LIN {X 0,Y 625.724,Z 847.824,A -85,B 0,C 180,E1 -6603.018,E2 -6603.018} C_VEL
LIN {X 0,Y 627.181,Z 825.978,A -85,B 0,C 180,E1 -6603.807,E2 -6603.807} C_VEL
LIN {X 0,Y 628.649,Z 801.844,A -85,B 0,C 180,E1 -6604.509,E2 -6604.509} C_VEL
LIN {X 0,Y 629.711,Z 779.175,A -85,B 0,C 180,E1 -6605.002,E2 -6605.002} C_VEL
LIN {X 0,Y 630.485,Z 755.504,A -85,B 0,C 180,E1 -6605.381,E2 -6605.381} C_VEL
LIN {X 0,Y 634.655,Z 505.847,A -85,B 0,C 180,E1 -6608.568,E2 -6608.568} C_VEL
LIN {X 0,Y 636.212,Z 410.489,A -85,B 0,C 180,E1 -6609.813,E2 -6609.813} C_VEL
LIN {X 0,Y 632.38,Z 394.65,A -85,B 0,C 180,E1 -6610.331,E2 -6610.331} C_VEL
LIN {X 0,Y 620.426,Z 374.094,A -85,B 0,C 180,E1 -6611.604,E2 -6611.604} C_VEL
LIN {X 0,Y 613.158,Z 355.776,A -85,B 0,C 180,E1 -6613.881,E2 -6613.881} C_VEL
LIN {X 0,Y 609.05,Z 345.363,A -85,B 0,C 180,E1 -6615.266,E2 -6615.266} C_VEL
LIN {X 0,Y 609.013,Z 345.362,A -85,B 0,C 180,E1 -6618.196,E2 -6618.196} C_VEL
LIN {X 0,Y 609.063,Z 345.362,A -85,B 0,C 180,E1 -6621.282,E2 -6621.282} C_VEL
LIN {X 0,Y 609.006,Z 345.32,A -85,B 0,C 180,E1 -6624.232,E2 -6624.232} C_VEL
LIN {X 0,Y 609.058,Z 345.363,A -85,B 0,C 180,E1 -6627.42,E2 -6627.42} C_VEL
LIN {X 0,Y 609.014,Z 345.363,A -85,B 0,C 180,E1 -6630.384,E2 -6630.384} C_VEL
LIN {X 0,Y 609.063,Z 345.359,A -85,B 0,C 180,E1 -6633.478,E2 -6633.478} C_VEL
LIN {X 0,Y 609.014,Z 345.358,A -85,B 0,C 180,E1 -6636.487,E2 -6636.487} C_VEL
LIN {X 0,Y 609.057,Z 345.353,A -85,B 0,C 180,E1 -6639.632,E2 -6639.632} C_VEL
LIN {X 0,Y 609.015,Z 345.363,A -85,B 0,C 180,E1 -6642.614,E2 -6642.614} C_VEL
LIN {X 0,Y 609.06,Z 345.366,A -85,B 0,C 180,E1 -6645.744,E2 -6645.744} C_VEL
LIN {X 0,Y 609.015,Z 345.354,A -85,B 0,C 180,E1 -6648.733,E2 -6648.733} C_VEL
LIN {X 0,Y 609.056,Z 345.352,A -85,B 0,C 180,E1 -6651.883,E2 -6651.883} C_VEL
LIN {X 0,Y 609.017,Z 345.364,A -85,B 0,C 180,E1 -6654.819,E2 -6654.819} C_VEL
LIN {X 0,Y 609.05,Z 345.354,A -85,B 0,C 180,E1 -6658.024,E2 -6658.024} C_VEL
LIN {X 0,Y 609.018,Z 345.36,A -85,B 0,C 180,E1 -6660.962,E2 -6660.962} C_VEL
LIN {X 0,Y 609.05,Z 345.368,A -85,B 0,C 180,E1 -6664.142,E2 -6664.142} C_VEL
LIN {X 0,Y 609.017,Z 345.351,A -85,B 0,C 180,E1 -6667.073,E2 -6667.073} C_VEL
LIN {X 0,Y 609.043,Z 345.356,A -85,B 0,C 180,E1 -6670.309,E2 -6670.309} C_VEL
LIN {X 0,Y 609.027,Z 345.363,A -85,B 0,C 180,E1 -6673.288,E2 -6673.288} C_VEL
LIN {X 0,Y 609.029,Z 345.361,A -85,B 0,C 180,E1 -6676.599,E2 -6676.599} C_VEL
LIN {X 0,Y 609.043,Z 345.358,A -85,B 0,C 180,E1 -6679.567,E2 -6679.567} C_VEL
LIN {X 0,Y 609.023,Z 345.362,A -85,B 0,C 180,E1 -6682.797,E2 -6682.797} C_VEL
LIN {X 0,Y 609.053,Z 345.361,A -85,B 0,C 180,E1 -6685.789,E2 -6685.789} C_VEL
LIN {X 0,Y 609.022,Z 345.367,A -85,B 0,C 180,E1 -6688.969,E2 -6688.969} C_VEL
LIN {X 0,Y 609.056,Z 345.351,A -85,B 0,C 180,E1 -6691.923,E2 -6691.923} C_VEL
LIN {X 0,Y 609.021,Z 345.362,A -85,B 0,C 180,E1 -6695.074,E2 -6695.074} C_VEL
LIN {X 0,Y 609.07,Z 345.352,A -85,B 0,C 180,E1 -6698.154,E2 -6698.154} C_VEL
LIN {X 0,Y 609.02,Z 345.37,A -85,B 0,C 180,E1 -6701.301,E2 -6701.301} C_VEL
LIN {X 0,Y 609.078,Z 345.362,A -85,B 0,C 180,E1 -6704.429,E2 -6704.429} C_VEL
LIN {X 0,Y 609.068,Z 345.578,A -85,B 0,C 180,E1 -6707.031,E2 -6707.031} C_VEL
LIN {X 0,Y 611.046,Z 350.8,A -85,B 0,C 180,E1 -6707.701,E2 -6707.701} C_VEL
LIN {X 0,Y 624.951,Z 372.362,A -85,B 0,C 180,E1 -6709.181,E2 -6709.181} C_VEL
LIN {X 0,Y 636.425,Z 391.644,A -85,B 0,C 180,E1 -6710.353,E2 -6710.353} C_VEL
LIN {X 0,Y 635.55,Z 441.225,A -85,B 0,C 180,E1 -6710.999,E2 -6710.999} C_VEL
LIN {X 0,Y 634.674,Z 448.921,A -85,B 0,C 180,E1 -6711.044,E2 -6711.044} C_VEL
LIN {X 0,Y 629.403,Z 469.491,A -85,B 0,C 180,E1 -6710.95,E2 -6710.95} C_VEL
LIN {X 0,Y 628.688,Z 476.1,A -85,B 0,C 180,E1 -6710.992,E2 -6710.992} C_VEL
LIN {X 0,Y 624.153,Z 726.916,A -85,B 0,C 180,E1 -6714.229,E2 -6714.229} C_VEL
LIN {X 0,Y 623.344,Z 751.398,A -85,B 0,C 180,E1 -6714.622,E2 -6714.622} C_VEL
LIN {X 0,Y 622.243,Z 774.459,A -85,B 0,C 180,E1 -6715.131,E2 -6715.131} C_VEL
LIN {X 0,Y 620.781,Z 797.913,A -85,B 0,C 180,E1 -6715.825,E2 -6715.825} C_VEL
LIN {X 0,Y 619.291,Z 818.986,A -85,B 0,C 180,E1 -6716.594,E2 -6716.594} C_VEL
LIN {X 0,Y 617.333,Z 842.509,A -85,B 0,C 180,E1 -6717.635,E2 -6717.635} C_VEL
LIN {X 0,Y 615.596,Z 861.479,A -85,B 0,C 180,E1 -6718.629,E2 -6718.629} C_VEL
LIN {X 0,Y 613.582,Z 882.127,A -85,B 0,C 180,E1 -6719.873,E2 -6719.873} C_VEL
LIN {X 0,Y 611.515,Z 901.861,A -85,B 0,C 180,E1 -6721.268,E2 -6721.268} C_VEL
LIN {X 0,Y 609.523,Z 921.125,A -85,B 0,C 180,E1 -6722.815,E2 -6722.815} C_VEL
LIN {X 0,Y 607.551,Z 939.267,A -85,B 0,C 180,E1 -6724.509,E2 -6724.509} C_VEL
LIN {X 0,Y 605.872,Z 955.81,A -85,B 0,C 180,E1 -6726.254,E2 -6726.254} C_VEL
LIN {X 0,Y 604.297,Z 971.472,A -85,B 0,C 180,E1 -6728.164,E2 -6728.164} C_VEL
LIN {X 0,Y 602.991,Z 986.499,A -85,B 0,C 180,E1 -6730.228,E2 -6730.228} C_VEL
LIN {X 0,Y 601.969,Z 999.427,A -85,B 0,C 180,E1 -6732.304,E2 -6732.304} C_VEL
LIN {X 0,Y 601.21,Z 1010.682,A -85,B 0,C 180,E1 -6734.37,E2 -6734.37} C_VEL
LIN {X 0,Y 600.63,Z 1020.967,A -85,B 0,C 180,E1 -6736.621,E2 -6736.621} C_VEL
LIN {X 0,Y 600.302,Z 1028.497,A -85,B 0,C 180,E1 -6738.568,E2 -6738.568} C_VEL
LIN {X 0,Y 600.056,Z 1036.101,A -85,B 0,C 180,E1 -6740.988,E2 -6740.988} C_VEL
LIN {X 0,Y 599.974,Z 1041.005,A -85,B 0,C 180,E1 -6743.012,E2 -6743.012} C_VEL
LIN {X 0,Y 599.921,Z 1045.157,A -85,B 0,C 180,E1 -6745.316,E2 -6745.316} C_VEL
LIN {X 0,Y 599.899,Z 1047.463,A -85,B 0,C 180,E1 -6747.516,E2 -6747.516} C_VEL
LIN {X 0,Y 599.894,Z 1048.384,A -85,B 0,C 180,E1 -6749.523,E2 -6749.523} C_VEL
LIN {X 0,Y 599.908,Z 1047.935,A -85,B 0,C 180,E1 -6751.91,E2 -6751.91} C_VEL
LIN {X 0,Y 599.919,Z 1046.062,A -85,B 0,C 180,E1 -6754.014,E2 -6754.014} C_VEL
LIN {X 0,Y 599.948,Z 1042.77,A -85,B 0,C 180,E1 -6756.219,E2 -6756.219} C_VEL
LIN {X 0,Y 600.026,Z 1037.609,A -85,B 0,C 180,E1 -6758.529,E2 -6758.529} C_VEL
LIN {X 0,Y 600.186,Z 1032.047,A -85,B 0,C 180,E1 -6760.462,E2 -6760.462} C_VEL
LIN {X 0,Y 600.514,Z 1023.769,A -85,B 0,C 180,E1 -6762.794,E2 -6762.794} C_VEL
LIN {X 0,Y 600.963,Z 1014.847,A -85,B 0,C 180,E1 -6764.846,E2 -6764.846} C_VEL
LIN {X 0,Y 601.657,Z 1003.931,A -85,B 0,C 180,E1 -6767.007,E2 -6767.007} C_VEL
LIN {X 0,Y 602.568,Z 991.521,A -85,B 0,C 180,E1 -6769.081,E2 -6769.081} C_VEL
LIN {X 0,Y 603.644,Z 978.717,A -85,B 0,C 180,E1 -6770.964,E2 -6770.964} C_VEL
LIN {X 0,Y 605.162,Z 962.65,A -85,B 0,C 180,E1 -6773.027,E2 -6773.027} C_VEL
LIN {X 0,Y 606.722,Z 947.311,A -85,B 0,C 180,E1 -6774.761,E2 -6774.761} C_VEL
LIN {X 0,Y 608.619,Z 929.224,A -85,B 0,C 180,E1 -6776.543,E2 -6776.543} C_VEL
LIN {X 0,Y 610.398,Z 912.383,A -85,B 0,C 180,E1 -6778.001,E2 -6778.001} C_VEL
LIN {X 0,Y 612.623,Z 891.447,A -85,B 0,C 180,E1 -6779.58,E2 -6779.58} C_VEL
LIN {X 0,Y 614.454,Z 873.223,A -85,B 0,C 180,E1 -6780.772,E2 -6780.772} C_VEL
LIN {X 0,Y 616.495,Z 852.089,A -85,B 0,C 180,E1 -6781.978,E2 -6781.978} C_VEL
LIN {X 0,Y 618.343,Z 830.28,A -85,B 0,C 180,E1 -6783.021,E2 -6783.021} C_VEL
LIN {X 0,Y 620.188,Z 807.62,A -85,B 0,C 180,E1 -6783.934,E2 -6783.934} C_VEL
LIN {X 0,Y 621.651,Z 784.687,A -85,B 0,C 180,E1 -6784.673,E2 -6784.673} C_VEL
LIN {X 0,Y 622.771,Z 764.523,A -85,B 0,C 180,E1 -6785.194,E2 -6785.194} C_VEL
LIN {X 0,Y 623.81,Z 738.844,A -85,B 0,C 180,E1 -6785.687,E2 -6785.687} C_VEL
LIN {X 0,Y 626.912,Z 571.696,A -85,B 0,C 180,E1 -6787.857,E2 -6787.857} C_VEL
LIN {X 0,Y 630.13,Z 394.451,A -85,B 0,C 180,E1 -6790.178,E2 -6790.178} C_VEL
LIN {X 0,Y 615.732,Z 370.831,A -85,B 0,C 180,E1 -6791.686,E2 -6791.686} C_VEL
LIN {X 0,Y 604.597,Z 353.811,A -85,B 0,C 180,E1 -6792.909,E2 -6792.909} C_VEL
LIN {X 0,Y 602.598,Z 350.289,A -85,B 0,C 180,E1 -6793.175,E2 -6793.175} C_VEL
LIN {X 0,Y 601.123,Z 346.314,A -85,B 0,C 180,E1 -6793.754,E2 -6793.754} C_VEL
LIN {X 0,Y 601.075,Z 346.354,A -85,B 0,C 180,E1 -6796.77,E2 -6796.77} C_VEL
LIN {X 0,Y 601.117,Z 346.328,A -85,B 0,C 180,E1 -6799.929,E2 -6799.929} C_VEL
LIN {X 0,Y 601.074,Z 346.348,A -85,B 0,C 180,E1 -6802.853,E2 -6802.853} C_VEL
LIN {X 0,Y 601.122,Z 346.344,A -85,B 0,C 180,E1 -6806.02,E2 -6806.02} C_VEL
LIN {X 0,Y 601.074,Z 346.347,A -85,B 0,C 180,E1 -6808.956,E2 -6808.956} C_VEL
LIN {X 0,Y 601.131,Z 346.339,A -85,B 0,C 180,E1 -6812.036,E2 -6812.036} C_VEL
LIN {X 0,Y 601.073,Z 346.356,A -85,B 0,C 180,E1 -6815.041,E2 -6815.041} C_VEL
LIN {X 0,Y 601.12,Z 346.352,A -85,B 0,C 180,E1 -6818.227,E2 -6818.227} C_VEL
LIN {X 0,Y 601.074,Z 346.346,A -85,B 0,C 180,E1 -6821.18,E2 -6821.18} C_VEL
LIN {X 0,Y 601.111,Z 346.337,A -85,B 0,C 180,E1 -6824.389,E2 -6824.389} C_VEL
LIN {X 0,Y 601.075,Z 346.356,A -85,B 0,C 180,E1 -6827.315,E2 -6827.315} C_VEL
LIN {X 0,Y 601.106,Z 346.352,A -85,B 0,C 180,E1 -6830.542,E2 -6830.542} C_VEL
LIN {X 0,Y 601.077,Z 346.344,A -85,B 0,C 180,E1 -6833.505,E2 -6833.505} C_VEL
LIN {X 0,Y 601.094,Z 346.35,A -85,B 0,C 180,E1 -6836.758,E2 -6836.758} C_VEL
LIN {X 0,Y 601.085,Z 346.347,A -85,B 0,C 180,E1 -6839.714,E2 -6839.714} C_VEL
LIN {X 0,Y 601.078,Z 346.336,A -85,B 0,C 180,E1 -6843.051,E2 -6843.051} C_VEL
LIN {X 0,Y 601.104,Z 346.357,A -85,B 0,C 180,E1 -6846.015,E2 -6846.015} C_VEL
LIN {X 0,Y 601.078,Z 346.352,A -85,B 0,C 180,E1 -6849.189,E2 -6849.189} C_VEL
LIN {X 0,Y 601.11,Z 346.341,A -85,B 0,C 180,E1 -6852.196,E2 -6852.196} C_VEL
LIN {X 0,Y 601.075,Z 346.351,A -85,B 0,C 180,E1 -6855.337,E2 -6855.337} C_VEL
LIN {X 0,Y 601.113,Z 346.351,A -85,B 0,C 180,E1 -6858.324,E2 -6858.324} C_VEL
LIN {X 0,Y 601.074,Z 346.348,A -85,B 0,C 180,E1 -6861.467,E2 -6861.467} C_VEL
LIN {X 0,Y 601.106,Z 346.343,A -85,B 0,C 180,E1 -6864.364,E2 -6864.364} C_VEL
LIN {X 0,Y 601.076,Z 346.348,A -85,B 0,C 180,E1 -6867.546,E2 -6867.546} C_VEL
LIN {X 0,Y 601.111,Z 346.351,A -85,B 0,C 180,E1 -6870.498,E2 -6870.498} C_VEL
LIN {X 0,Y 601.076,Z 346.354,A -85,B 0,C 180,E1 -6873.638,E2 -6873.638} C_VEL
LIN {X 0,Y 601.117,Z 346.348,A -85,B 0,C 180,E1 -6876.667,E2 -6876.667} C_VEL
LIN {X 0,Y 601.07,Z 346.333,A -85,B 0,C 180,E1 -6879.826,E2 -6879.826} C_VEL
LIN {X 0,Y 601.127,Z 346.352,A -85,B 0,C 180,E1 -6882.868,E2 -6882.868} C_VEL
LIN {X 0,Y 601.073,Z 346.369,A -85,B 0,C 180,E1 -6884.115,E2 -6884.115} C_VEL
LIN {X 0,Y 602.516,Z 349.999,A -85,B 0,C 180,E1 -6884.607,E2 -6884.607} C_VEL
LIN {X 0,Y 610.857,Z 370.649,A -85,B 0,C 180,E1 -6887.304,E2 -6887.304} C_VEL
LIN {X 0,Y 612.529,Z 374.694,A -85,B 0,C 180,E1 -6887.774,E2 -6887.774} C_VEL
LIN {X 0,Y 627.059,Z 399.331,A -85,B 0,C 180,E1 -6889.325,E2 -6889.325} C_VEL
LIN {X 0,Y 630.151,Z 413.759,A -85,B 0,C 180,E1 -6889.776,E2 -6889.776} C_VEL
LIN {X 0,Y 625.275,Z 679.186,A -85,B 0,C 180,E1 -6893.217,E2 -6893.217} C_VEL
LIN {X 0,Y 623.608,Z 766.862,A -85,B 0,C 180,E1 -6894.36,E2 -6894.36} C_VEL
LIN {X 0,Y 622.517,Z 792.121,A -85,B 0,C 180,E1 -6894.846,E2 -6894.846} C_VEL
LIN {X 0,Y 621.337,Z 812.739,A -85,B 0,C 180,E1 -6895.377,E2 -6895.377} C_VEL
LIN {X 0,Y 619.82,Z 835.991,A -85,B 0,C 180,E1 -6896.127,E2 -6896.127} C_VEL
LIN {X 0,Y 618.034,Z 858.17,A -85,B 0,C 180,E1 -6897.016,E2 -6897.016} C_VEL
LIN {X 0,Y 616.225,Z 879.509,A -85,B 0,C 180,E1 -6898.025,E2 -6898.025} C_VEL
LIN {X 0,Y 614.17,Z 901.39,A -85,B 0,C 180,E1 -6899.256,E2 -6899.256} C_VEL
LIN {X 0,Y 612.363,Z 919.938,A -85,B 0,C 180,E1 -6900.454,E2 -6900.454} C_VEL
LIN {X 0,Y 610.172,Z 941.383,A -85,B 0,C 180,E1 -6902.052,E2 -6902.052} C_VEL
LIN {X 0,Y 608.468,Z 958.211,A -85,B 0,C 180,E1 -6903.487,E2 -6903.487} C_VEL
LIN {X 0,Y 606.561,Z 977.391,A -85,B 0,C 180,E1 -6905.351,E2 -6905.351} C_VEL
LIN {X 0,Y 605.094,Z 992.652,A -85,B 0,C 180,E1 -6907.047,E2 -6907.047} C_VEL
LIN {X 0,Y 603.75,Z 1007.707,A -85,B 0,C 180,E1 -6908.938,E2 -6908.938} C_VEL
LIN {X 0,Y 602.59,Z 1021.237,A -85,B 0,C 180,E1 -6910.92,E2 -6910.92} C_VEL
LIN {X 0,Y 601.668,Z 1033.688,A -85,B 0,C 180,E1 -6912.993,E2 -6912.993} C_VEL
LIN {X 0,Y 600.962,Z 1044.707,A -85,B 0,C 180,E1 -6915.168,E2 -6915.168} C_VEL
LIN {X 0,Y 600.516,Z 1053.583,A -85,B 0,C 180,E1 -6917.206,E2 -6917.206} C_VEL
LIN {X 0,Y 600.189,Z 1061.907,A -85,B 0,C 180,E1 -6919.538,E2 -6919.538} C_VEL
LIN {X 0,Y 600.028,Z 1067.491,A -85,B 0,C 180,E1 -6921.471,E2 -6921.471} C_VEL
LIN {X 0,Y 599.946,Z 1072.695,A -85,B 0,C 180,E1 -6923.781,E2 -6923.781} C_VEL
LIN {X 0,Y 599.911,Z 1076.009,A -85,B 0,C 180,E1 -6925.986,E2 -6925.986} C_VEL
LIN {X 0,Y 599.906,Z 1077.835,A -85,B 0,C 180,E1 -6927.994,E2 -6927.994} C_VEL
LIN {X 0,Y 599.895,Z 1078.417,A -85,B 0,C 180,E1 -6930.382,E2 -6930.382} C_VEL
LIN {X 0,Y 599.908,Z 1077.495,A -85,B 0,C 180,E1 -6932.484,E2 -6932.484} C_VEL
LIN {X 0,Y 599.925,Z 1075.085,A -85,B 0,C 180,E1 -6934.78,E2 -6934.78} C_VEL
LIN {X 0,Y 599.968,Z 1071.102,A -85,B 0,C 180,E1 -6936.988,E2 -6936.988} C_VEL
LIN {X 0,Y 600.05,Z 1066.22,A -85,B 0,C 180,E1 -6939.012,E2 -6939.012} C_VEL
LIN {X 0,Y 600.302,Z 1058.66,A -85,B 0,C 180,E1 -6941.432,E2 -6941.432} C_VEL
LIN {X 0,Y 600.649,Z 1050.748,A -85,B 0,C 180,E1 -6943.477,E2 -6943.477} C_VEL
LIN {X 0,Y 601.23,Z 1040.401,A -85,B 0,C 180,E1 -6945.729,E2 -6945.729} C_VEL
LIN {X 0,Y 601.99,Z 1029.112,A -85,B 0,C 180,E1 -6947.795,E2 -6947.795} C_VEL
LIN {X 0,Y 603.058,Z 1015.704,A -85,B 0,C 180,E1 -6949.93,E2 -6949.93} C_VEL
LIN {X 0,Y 604.209,Z 1002.366,A -85,B 0,C 180,E1 -6951.758,E2 -6951.758} C_VEL
LIN {X 0,Y 605.684,Z 986.674,A -85,B 0,C 180,E1 -6953.65,E2 -6953.65} C_VEL
LIN {X 0,Y 607.335,Z 969.48,A -85,B 0,C 180,E1 -6955.448,E2 -6955.448} C_VEL
LIN {X 0,Y 609.03,Z 952.777,A -85,B 0,C 180,E1 -6956.997,E2 -6956.997} C_VEL
LIN {X 0,Y 611.098,Z 932.379,A -85,B 0,C 180,E1 -6958.647,E2 -6958.647} C_VEL
LIN {X 0,Y 612.925,Z 914.012,A -85,B 0,C 180,E1 -6959.946,E2 -6959.946} C_VEL
LIN {X 0,Y 615.152,Z 891.168,A -85,B 0,C 180,E1 -6961.341,E2 -6961.341} C_VEL
LIN {X 0,Y 616.861,Z 872.159,A -85,B 0,C 180,E1 -6962.338,E2 -6962.338} C_VEL
LIN {X 0,Y 618.757,Z 849.987,A -85,B 0,C 180,E1 -6963.336,E2 -6963.336} C_VEL
LIN {X 0,Y 620.364,Z 827.247,A -85,B 0,C 180,E1 -6964.174,E2 -6964.174} C_VEL
LIN {X 0,Y 621.87,Z 804.068,A -85,B 0,C 180,E1 -6964.869,E2 -6964.869} C_VEL
LIN {X 0,Y 623.089,Z 780.098,A -85,B 0,C 180,E1 -6965.405,E2 -6965.405} C_VEL
LIN {X 0,Y 623.875,Z 757.874,A -85,B 0,C 180,E1 -6965.77,E2 -6965.77} C_VEL
LIN {X 0,Y 628.256,Z 512.479,A -85,B 0,C 180,E1 -6968.937,E2 -6968.937} C_VEL
LIN {X 0,Y 629.985,Z 412.169,A -85,B 0,C 180,E1 -6970.259,E2 -6970.259} C_VEL
LIN {X 0,Y 626.717,Z 398.735,A -85,B 0,C 180,E1 -6970.708,E2 -6970.708} C_VEL
LIN {X 0,Y 612.172,Z 373.992,A -85,B 0,C 180,E1 -6972.276,E2 -6972.276} C_VEL
LIN {X 0,Y 605.295,Z 356.861,A -85,B 0,C 180,E1 -6974.469,E2 -6974.469} C_VEL
LIN {X 0,Y 602.041,Z 349.262,A -85,B 0,C 180,E1 -6975.503,E2 -6975.503} C_VEL
LIN {X 0,Y 601.072,Z 346.353,A -85,B 0,C 180,E1 -6975.885,E2 -6975.885} C_VEL
LIN {X 0,Y 601.145,Z 346.353,A -85,B 0,C 180,E1 -6979.054,E2 -6979.054} C_VEL
LIN {X 0,Y 601.071,Z 346.354,A -85,B 0,C 180,E1 -6982.132,E2 -6982.132} C_VEL
LIN {X 0,Y 601.127,Z 346.308,A -85,B 0,C 180,E1 -6985.255,E2 -6985.255} C_VEL
LIN {X 0,Y 601.071,Z 346.347,A -85,B 0,C 180,E1 -6988.286,E2 -6988.286} C_VEL
LIN {X 0,Y 601.134,Z 346.343,A -85,B 0,C 180,E1 -6991.377,E2 -6991.377} C_VEL
LIN {X 0,Y 601.078,Z 346.353,A -85,B 0,C 180,E1 -6994.479,E2 -6994.479} C_VEL
LIN {X 0,Y 601.108,Z 346.357,A -85,B 0,C 180,E1 -6997.712,E2 -6997.712} C_VEL
LIN {X 0,Y 601.079,Z 346.348,A -85,B 0,C 180,E1 -7000.668,E2 -7000.668} C_VEL
LIN {X 0,Y 601.091,Z 346.343,A -85,B 0,C 180,E1 -7003.97,E2 -7003.97} C_VEL
LIN {X 0,Y 601.085,Z 346.352,A -85,B 0,C 180,E1 -7006.827,E2 -7006.827} C_VEL
LIN {X 0,Y 601.087,Z 346.357,A -85,B 0,C 180,E1 -7010.134,E2 -7010.134} C_VEL
LIN {X 0,Y 601.089,Z 346.336,A -85,B 0,C 180,E1 -7013.025,E2 -7013.025} C_VEL
LIN {X 0,Y 601.085,Z 346.346,A -85,B 0,C 180,E1 -7016.28,E2 -7016.28} C_VEL
LIN {X 0,Y 601.101,Z 346.35,A -85,B 0,C 180,E1 -7019.238,E2 -7019.238} C_VEL
LIN {X 0,Y 601.08,Z 346.345,A -85,B 0,C 180,E1 -7022.479,E2 -7022.479} C_VEL
LIN {X 0,Y 601.123,Z 346.351,A -85,B 0,C 180,E1 -7025.536,E2 -7025.536} C_VEL
LIN {X 0,Y 601.077,Z 346.355,A -85,B 0,C 180,E1 -7028.707,E2 -7028.707} C_VEL
LIN {X 0,Y 601.134,Z 346.335,A -85,B 0,C 180,E1 -7031.806,E2 -7031.806} C_VEL
LIN {X 0,Y 601.075,Z 346.347,A -85,B 0,C 180,E1 -7034.942,E2 -7034.942} C_VEL
LIN {X 0,Y 601.14,Z 346.351,A -85,B 0,C 180,E1 -7038.022,E2 -7038.022} C_VEL
LIN {X 0,Y 601.077,Z 346.352,A -85,B 0,C 180,E1 -7041.058,E2 -7041.058} C_VEL
LIN {X 0,Y 601.138,Z 346.339,A -85,B 0,C 180,E1 -7044.153,E2 -7044.153} C_VEL
LIN {X 0,Y 601.077,Z 346.347,A -85,B 0,C 180,E1 -7047.224,E2 -7047.224} C_VEL
LIN {X 0,Y 601.14,Z 346.346,A -85,B 0,C 180,E1 -7050.375,E2 -7050.375} C_VEL
LIN {X 0,Y 601.079,Z 346.353,A -85,B 0,C 180,E1 -7053.409,E2 -7053.409} C_VEL
LIN {X 0,Y 601.131,Z 346.35,A -85,B 0,C 180,E1 -7056.547,E2 -7056.547} C_VEL
LIN {X 0,Y 601.084,Z 346.354,A -85,B 0,C 180,E1 -7059.629,E2 -7059.629} C_VEL
LIN {X 0,Y 601.108,Z 346.348,A -85,B 0,C 180,E1 -7062.87,E2 -7062.87} C_VEL
LIN {X 0,Y 601.09,Z 346.354,A -85,B 0,C 180,E1 -7065.814,E2 -7065.814} C_VEL
LIN {X 0,Y 601.149,Z 346.434,A -85,B 0,C 180,E1 -7066.383,E2 -7066.383} C_VEL
LIN {X 0,Y 602.873,Z 351.044,A -85,B 0,C 180,E1 -7066.988,E2 -7066.988} C_VEL
LIN {X 0,Y 616.862,Z 372.628,A -85,B 0,C 180,E1 -7068.528,E2 -7068.528} C_VEL
LIN {X 0,Y 630.226,Z 394.791,A -85,B 0,C 180,E1 -7069.926,E2 -7069.926} C_VEL
LIN {X 0,Y 628.688,Z 476.1,A -85,B 0,C 180,E1 -7070.992,E2 -7070.992} C_VEL
LIN {X 0,Y 627.774,Z 483.796,A -85,B 0,C 180,E1 -7071.035,E2 -7071.035} C_VEL
LIN {X 0,Y 622.511,Z 504.356,A -85,B 0,C 180,E1 -7070.94,E2 -7070.94} C_VEL
LIN {X 0,Y 621.779,Z 510.962,A -85,B 0,C 180,E1 -7070.981,E2 -7070.981} C_VEL
LIN {X 0,Y 617.332,Z 738.525,A -85,B 0,C 180,E1 -7073.962,E2 -7073.962} C_VEL
LIN {X 0,Y 616.243,Z 764.43,A -85,B 0,C 180,E1 -7074.459,E2 -7074.459} C_VEL
LIN {X 0,Y 615.067,Z 784.637,A -85,B 0,C 180,E1 -7074.984,E2 -7074.984} C_VEL
LIN {X 0,Y 613.562,Z 807.208,A -85,B 0,C 180,E1 -7075.714,E2 -7075.714} C_VEL
LIN {X 0,Y 611.658,Z 829.758,A -85,B 0,C 180,E1 -7076.625,E2 -7076.625} C_VEL
LIN {X 0,Y 609.851,Z 849.73,A -85,B 0,C 180,E1 -7077.579,E2 -7077.579} C_VEL
LIN {X 0,Y 607.612,Z 872.056,A -85,B 0,C 180,E1 -7078.839,E2 -7078.839} C_VEL
LIN {X 0,Y 605.679,Z 890.202,A -85,B 0,C 180,E1 -7080.028,E2 -7080.028} C_VEL
LIN {X 0,Y 603.368,Z 911.11,A -85,B 0,C 180,E1 -7081.601,E2 -7081.601} C_VEL
LIN {X 0,Y 601.376,Z 928.51,A -85,B 0,C 180,E1 -7083.112,E2 -7083.112} C_VEL
LIN {X 0,Y 599.464,Z 945.958,A -85,B 0,C 180,E1 -7084.828,E2 -7084.828} C_VEL
LIN {X 0,Y 597.694,Z 961.932,A -85,B 0,C 180,E1 -7086.642,E2 -7086.642} C_VEL
LIN {X 0,Y 596.188,Z 976.928,A -85,B 0,C 180,E1 -7088.563,E2 -7088.563} C_VEL
LIN {X 0,Y 594.877,Z 990.364,A -85,B 0,C 180,E1 -7090.561,E2 -7090.561} C_VEL
LIN {X 0,Y 593.84,Z 1003.442,A -85,B 0,C 180,E1 -7092.762,E2 -7092.762} C_VEL
LIN {X 0,Y 593.08,Z 1014.434,A -85,B 0,C 180,E1 -7094.952,E2 -7094.952} C_VEL
LIN {X 0,Y 592.582,Z 1023.397,A -85,B 0,C 180,E1 -7097.032,E2 -7097.032} C_VEL
LIN {X 0,Y 592.222,Z 1031.767,A -85,B 0,C 180,E1 -7099.395,E2 -7099.395} C_VEL
LIN {X 0,Y 592.038,Z 1037.374,A -85,B 0,C 180,E1 -7101.355,E2 -7101.355} C_VEL
LIN {X 0,Y 591.952,Z 1042.621,A -85,B 0,C 180,E1 -7103.697,E2 -7103.697} C_VEL
LIN {X 0,Y 591.92,Z 1045.955,A -85,B 0,C 180,E1 -7105.932,E2 -7105.932} C_VEL
LIN {X 0,Y 591.91,Z 1047.803,A -85,B 0,C 180,E1 -7107.967,E2 -7107.967} C_VEL
LIN {X 0,Y 591.895,Z 1048.427,A -85,B 0,C 180,E1 -7110.387,E2 -7110.387} C_VEL
LIN {X 0,Y 591.907,Z 1047.594,A -85,B 0,C 180,E1 -7112.42,E2 -7112.42} C_VEL
LIN {X 0,Y 591.922,Z 1045.493,A -85,B 0,C 180,E1 -7114.554,E2 -7114.554} C_VEL
LIN {X 0,Y 591.97,Z 1041.404,A -85,B 0,C 180,E1 -7116.985,E2 -7116.985} C_VEL
LIN {X 0,Y 592.055,Z 1036.59,A -85,B 0,C 180,E1 -7119.037,E2 -7119.037} C_VEL
LIN {X 0,Y 592.3,Z 1029.528,A -85,B 0,C 180,E1 -7121.392,E2 -7121.392} C_VEL
LIN {X 0,Y 592.654,Z 1021.74,A -85,B 0,C 180,E1 -7123.464,E2 -7123.464} C_VEL
LIN {X 0,Y 593.231,Z 1012.089,A -85,B 0,C 180,E1 -7125.645,E2 -7125.645} C_VEL
LIN {X 0,Y 594.056,Z 1000.505,A -85,B 0,C 180,E1 -7127.839,E2 -7127.839} C_VEL
LIN {X 0,Y 595.198,Z 987.15,A -85,B 0,C 180,E1 -7130.042,E2 -7130.042} C_VEL
LIN {X 0,Y 596.544,Z 972.961,A -85,B 0,C 180,E1 -7132.052,E2 -7132.052} C_VEL
LIN {X 0,Y 598.08,Z 958.467,A -85,B 0,C 180,E1 -7133.865,E2 -7133.865} C_VEL
LIN {X 0,Y 600.001,Z 940.845,A -85,B 0,C 180,E1 -7135.782,E2 -7135.782} C_VEL
LIN {X 0,Y 601.879,Z 924.287,A -85,B 0,C 180,E1 -7137.364,E2 -7137.364} C_VEL
LIN {X 0,Y 604.105,Z 904.517,A -85,B 0,C 180,E1 -7139.01,E2 -7139.01} C_VEL
LIN {X 0,Y 606.071,Z 886.477,A -85,B 0,C 180,E1 -7140.321,E2 -7140.321} C_VEL
LIN {X 0,Y 608.449,Z 864.055,A -85,B 0,C 180,E1 -7141.727,E2 -7141.727} C_VEL
LIN {X 0,Y 610.258,Z 845.342,A -85,B 0,C 180,E1 -7142.731,E2 -7142.731} C_VEL
LIN {X 0,Y 612.24,Z 823.731,A -85,B 0,C 180,E1 -7143.73,E2 -7143.73} C_VEL
LIN {X 0,Y 613.987,Z 800.484,A -85,B 0,C 180,E1 -7144.607,E2 -7144.607} C_VEL
LIN {X 0,Y 615.456,Z 778.397,A -85,B 0,C 180,E1 -7145.286,E2 -7145.286} C_VEL
LIN {X 0,Y 616.738,Z 753.691,A -85,B 0,C 180,E1 -7145.86,E2 -7145.86} C_VEL
LIN {X 0,Y 617.543,Z 731.585,A -85,B 0,C 180,E1 -7146.231,E2 -7146.231} C_VEL
LIN {X 0,Y 622.408,Z 480.872,A -85,B 0,C 180,E1 -7149.503,E2 -7149.503} C_VEL
LIN {X 0,Y 623.894,Z 397.629,A -85,B 0,C 180,E1 -7150.618,E2 -7150.618} C_VEL
LIN {X 0,Y 610.742,Z 375.972,A -85,B 0,C 180,E1 -7152.027,E2 -7152.027} C_VEL
LIN {X 0,Y 600.094,Z 359.572,A -85,B 0,C 180,E1 -7153.219,E2 -7153.219} C_VEL
LIN {X 0,Y 594.493,Z 350.816,A -85,B 0,C 180,E1 -7153.887,E2 -7153.887} C_VEL
LIN {X 0,Y 593.132,Z 347.309,A -85,B 0,C 180,E1 -7154.395,E2 -7154.395} C_VEL
LIN {X 0,Y 593.192,Z 347.311,A -85,B 0,C 180,E1 -7157.473,E2 -7157.473} C_VEL
LIN {X 0,Y 593.134,Z 347.341,A -85,B 0,C 180,E1 -7160.542,E2 -7160.542} C_VEL
LIN {X 0,Y 593.195,Z 347.336,A -85,B 0,C 180,E1 -7163.606,E2 -7163.606} C_VEL
LIN {X 0,Y 593.133,Z 347.343,A -85,B 0,C 180,E1 -7166.778,E2 -7166.778} C_VEL
LIN {X 0,Y 593.199,Z 347.337,A -85,B 0,C 180,E1 -7169.959,E2 -7169.959} C_VEL
LIN {X 0,Y 593.135,Z 347.333,A -85,B 0,C 180,E1 -7173.033,E2 -7173.033} C_VEL
LIN {X 0,Y 593.174,Z 347.328,A -85,B 0,C 180,E1 -7176.251,E2 -7176.251} C_VEL
LIN {X 0,Y 593.136,Z 347.345,A -85,B 0,C 180,E1 -7179.164,E2 -7179.164} C_VEL
LIN {X 0,Y 593.175,Z 347.341,A -85,B 0,C 180,E1 -7182.337,E2 -7182.337} C_VEL
LIN {X 0,Y 593.136,Z 347.332,A -85,B 0,C 180,E1 -7185.353,E2 -7185.353} C_VEL
LIN {X 0,Y 593.154,Z 347.327,A -85,B 0,C 180,E1 -7188.625,E2 -7188.625} C_VEL
LIN {X 0,Y 593.146,Z 347.345,A -85,B 0,C 180,E1 -7191.567,E2 -7191.567} C_VEL
LIN {X 0,Y 593.143,Z 347.339,A -85,B 0,C 180,E1 -7194.874,E2 -7194.874} C_VEL
LIN {X 0,Y 593.163,Z 347.332,A -85,B 0,C 180,E1 -7197.875,E2 -7197.875} C_VEL
LIN {X 0,Y 593.139,Z 347.343,A -85,B 0,C 180,E1 -7201.063,E2 -7201.063} C_VEL
LIN {X 0,Y 593.17,Z 347.329,A -85,B 0,C 180,E1 -7204.06,E2 -7204.06} C_VEL
LIN {X 0,Y 593.132,Z 347.333,A -85,B 0,C 180,E1 -7207.264,E2 -7207.264} C_VEL
LIN {X 0,Y 593.186,Z 347.343,A -85,B 0,C 180,E1 -7210.293,E2 -7210.293} C_VEL
LIN {X 0,Y 593.131,Z 347.339,A -85,B 0,C 180,E1 -7213.453,E2 -7213.453} C_VEL
LIN {X 0,Y 593.191,Z 347.326,A -85,B 0,C 180,E1 -7216.45,E2 -7216.45} C_VEL
LIN {X 0,Y 593.132,Z 347.341,A -85,B 0,C 180,E1 -7219.601,E2 -7219.601} C_VEL
LIN {X 0,Y 593.204,Z 347.339,A -85,B 0,C 180,E1 -7222.706,E2 -7222.706} C_VEL
LIN {X 0,Y 593.132,Z 347.342,A -85,B 0,C 180,E1 -7225.815,E2 -7225.815} C_VEL
LIN {X 0,Y 593.194,Z 347.337,A -85,B 0,C 180,E1 -7228.975,E2 -7228.975} C_VEL
LIN {X 0,Y 593.133,Z 347.339,A -85,B 0,C 180,E1 -7232.011,E2 -7232.011} C_VEL
LIN {X 0,Y 593.176,Z 347.341,A -85,B 0,C 180,E1 -7235.205,E2 -7235.205} C_VEL
LIN {X 0,Y 593.139,Z 347.346,A -85,B 0,C 180,E1 -7238.227,E2 -7238.227} C_VEL
LIN {X 0,Y 593.147,Z 347.31,A -85,B 0,C 180,E1 -7241.542,E2 -7241.542} C_VEL
LIN {X 0,Y 593.169,Z 347.375,A -85,B 0,C 180,E1 -7243.453,E2 -7243.453} C_VEL
LIN {X 0,Y 594.279,Z 350.575,A -85,B 0,C 180,E1 -7243.884,E2 -7243.884} C_VEL
LIN {X 0,Y 600.713,Z 365.835,A -85,B 0,C 180,E1 -7245.978,E2 -7245.978} C_VEL
LIN {X 0,Y 604.075,Z 374.283,A -85,B 0,C 180,E1 -7247.04,E2 -7247.04} C_VEL
LIN {X 0,Y 617.94,Z 397.22,A -85,B 0,C 180,E1 -7248.567,E2 -7248.567} C_VEL
LIN {X 0,Y 621.641,Z 404.242,A -85,B 0,C 180,E1 -7248.971,E2 -7248.971} C_VEL
LIN {X 0,Y 623.995,Z 415.473,A -85,B 0,C 180,E1 -7249.324,E2 -7249.324} C_VEL
LIN {X 0,Y 618.837,Z 680.262,A -85,B 0,C 180,E1 -7252.788,E2 -7252.788} C_VEL
LIN {X 0,Y 617.095,Z 766.739,A -85,B 0,C 180,E1 -7253.927,E2 -7253.927} C_VEL
LIN {X 0,Y 615.933,Z 792.104,A -85,B 0,C 180,E1 -7254.419,E2 -7254.419} C_VEL
LIN {X 0,Y 614.673,Z 812.984,A -85,B 0,C 180,E1 -7254.962,E2 -7254.962} C_VEL
LIN {X 0,Y 612.986,Z 837.065,A -85,B 0,C 180,E1 -7255.753,E2 -7255.753} C_VEL
LIN {X 0,Y 611.222,Z 857.953,A -85,B 0,C 180,E1 -7256.6,E2 -7256.6} C_VEL
LIN {X 0,Y 609.326,Z 879.005,A -85,B 0,C 180,E1 -7257.603,E2 -7257.603} C_VEL
LIN {X 0,Y 607.113,Z 901.171,A -85,B 0,C 180,E1 -7258.859,E2 -7258.859} C_VEL
LIN {X 0,Y 605.156,Z 920.182,A -85,B 0,C 180,E1 -7260.101,E2 -7260.101} C_VEL
LIN {X 0,Y 602.885,Z 941.163,A -85,B 0,C 180,E1 -7261.684,E2 -7261.684} C_VEL
LIN {X 0,Y 601.041,Z 958.154,A -85,B 0,C 180,E1 -7263.149,E2 -7263.149} C_VEL
LIN {X 0,Y 599.033,Z 977.169,A -85,B 0,C 180,E1 -7265.02,E2 -7265.02} C_VEL
LIN {X 0,Y 597.459,Z 992.43,A -85,B 0,C 180,E1 -7266.736,E2 -7266.736} C_VEL
LIN {X 0,Y 595.961,Z 1008.239,A -85,B 0,C 180,E1 -7268.752,E2 -7268.752} C_VEL
LIN {X 0,Y 594.797,Z 1021.223,A -85,B 0,C 180,E1 -7270.66,E2 -7270.66} C_VEL
LIN {X 0,Y 593.816,Z 1033.687,A -85,B 0,C 180,E1 -7272.761,E2 -7272.761} C_VEL
LIN {X 0,Y 593.06,Z 1044.636,A -85,B 0,C 180,E1 -7274.951,E2 -7274.951} C_VEL
LIN {X 0,Y 592.571,Z 1053.582,A -85,B 0,C 180,E1 -7277.031,E2 -7277.031} C_VEL
LIN {X 0,Y 592.218,Z 1061.906,A -85,B 0,C 180,E1 -7279.395,E2 -7279.395} C_VEL
LIN {X 0,Y 592.035,Z 1067.491,A -85,B 0,C 180,E1 -7281.355,E2 -7281.355} C_VEL
LIN {X 0,Y 591.946,Z 1072.695,A -85,B 0,C 180,E1 -7283.696,E2 -7283.696} C_VEL
LIN {X 0,Y 591.913,Z 1075.895,A -85,B 0,C 180,E1 -7285.834,E2 -7285.834} C_VEL
LIN {X 0,Y 591.909,Z 1077.767,A -85,B 0,C 180,E1 -7287.87,E2 -7287.87} C_VEL
LIN {X 0,Y 591.898,Z 1078.439,A -85,B 0,C 180,E1 -7290.29,E2 -7290.29} C_VEL
LIN {X 0,Y 591.909,Z 1077.562,A -85,B 0,C 180,E1 -7292.42,E2 -7292.42} C_VEL
LIN {X 0,Y 591.918,Z 1075.439,A -85,B 0,C 180,E1 -7294.554,E2 -7294.554} C_VEL
LIN {X 0,Y 591.97,Z 1071.308,A -85,B 0,C 180,E1 -7296.985,E2 -7296.985} C_VEL
LIN {X 0,Y 592.058,Z 1066.474,A -85,B 0,C 180,E1 -7299.036,E2 -7299.036} C_VEL
LIN {X 0,Y 592.31,Z 1059.366,A -85,B 0,C 180,E1 -7301.391,E2 -7301.391} C_VEL
LIN {X 0,Y 592.669,Z 1051.557,A -85,B 0,C 180,E1 -7303.463,E2 -7303.463} C_VEL
LIN {X 0,Y 593.246,Z 1041.888,A -85,B 0,C 180,E1 -7305.645,E2 -7305.645} C_VEL
LIN {X 0,Y 594.073,Z 1030.257,A -85,B 0,C 180,E1 -7307.838,E2 -7307.838} C_VEL
LIN {X 0,Y 594.957,Z 1019.298,A -85,B 0,C 180,E1 -7309.641,E2 -7309.641} C_VEL
LIN {X 0,Y 596.372,Z 1003.703,A -85,B 0,C 180,E1 -7311.852,E2 -7311.852} C_VEL
LIN {X 0,Y 597.72,Z 989.869,A -85,B 0,C 180,E1 -7313.566,E2 -7313.566} C_VEL
LIN {X 0,Y 599.552,Z 972.329,A -85,B 0,C 180,E1 -7315.485,E2 -7315.485} C_VEL
LIN {X 0,Y 601.341,Z 955.356,A -85,B 0,C 180,E1 -7317.103,E2 -7317.103} C_VEL
LIN {X 0,Y 603.459,Z 936.197,A -85,B 0,C 180,E1 -7318.719,E2 -7318.719} C_VEL
LIN {X 0,Y 605.49,Z 916.752,A -85,B 0,C 180,E1 -7320.133,E2 -7320.133} C_VEL
LIN {X 0,Y 607.638,Z 896.27,A -85,B 0,C 180,E1 -7321.442,E2 -7321.442} C_VEL
LIN {X 0,Y 609.722,Z 874.646,A -85,B 0,C 180,E1 -7322.614,E2 -7322.614} C_VEL
LIN {X 0,Y 611.481,Z 855.151,A -85,B 0,C 180,E1 -7323.522,E2 -7323.522} C_VEL
LIN {X 0,Y 613.478,Z 829.999,A -85,B 0,C 180,E1 -7324.498,E2 -7324.498} C_VEL
LIN {X 0,Y 614.932,Z 808.635,A -85,B 0,C 180,E1 -7325.164,E2 -7325.164} C_VEL
LIN {X 0,Y 616.39,Z 783.294,A -85,B 0,C 180,E1 -7325.774,E2 -7325.774} C_VEL
LIN {X 0,Y 617.278,Z 760.761,A -85,B 0,C 180,E1 -7326.161,E2 -7326.161} C_VEL
LIN {X 0,Y 621.819,Z 522.344,A -85,B 0,C 180,E1 -7329.27,E2 -7329.27} C_VEL
LIN {X 0,Y 623.833,Z 414.042,A -85,B 0,C 180,E1 -7330.708,E2 -7330.708} C_VEL
LIN {X 0,Y 621.166,Z 402.952,A -85,B 0,C 180,E1 -7331.084,E2 -7331.084} C_VEL
LIN {X 0,Y 606.973,Z 378.963,A -85,B 0,C 180,E1 -7332.63,E2 -7332.63} C_VEL
LIN {X 0,Y 603.682,Z 373.486,A -85,B 0,C 180,E1 -7333.032,E2 -7333.032} C_VEL
LIN {X 0,Y 596.242,Z 354.867,A -85,B 0,C 180,E1 -7335.494,E2 -7335.494} C_VEL
LIN {X 0,Y 593.191,Z 347.55,A -85,B 0,C 180,E1 -7336.519,E2 -7336.519} C_VEL
LIN {X 0,Y 593.137,Z 347.34,A -85,B 0,C 180,E1 -7339.787,E2 -7339.787} C_VEL
LIN {X 0,Y 593.174,Z 347.315,A -85,B 0,C 180,E1 -7342.76,E2 -7342.76} C_VEL
LIN {X 0,Y 593.133,Z 347.322,A -85,B 0,C 180,E1 -7345.966,E2 -7345.966} C_VEL
LIN {X 0,Y 593.199,Z 347.325,A -85,B 0,C 180,E1 -7349.089,E2 -7349.089} C_VEL
LIN {X 0,Y 593.133,Z 347.33,A -85,B 0,C 180,E1 -7352.163,E2 -7352.163} C_VEL
LIN {X 0,Y 593.201,Z 347.33,A -85,B 0,C 180,E1 -7355.303,E2 -7355.303} C_VEL
LIN {X 0,Y 593.134,Z 347.343,A -85,B 0,C 180,E1 -7358.335,E2 -7358.335} C_VEL
LIN {X 0,Y 593.2,Z 347.337,A -85,B 0,C 180,E1 -7361.423,E2 -7361.423} C_VEL
LIN {X 0,Y 593.135,Z 347.336,A -85,B 0,C 180,E1 -7364.553,E2 -7364.553} C_VEL
LIN {X 0,Y 593.182,Z 347.328,A -85,B 0,C 180,E1 -7367.737,E2 -7367.737} C_VEL
LIN {X 0,Y 593.14,Z 347.343,A -85,B 0,C 180,E1 -7370.785,E2 -7370.785} C_VEL
LIN {X 0,Y 593.166,Z 347.338,A -85,B 0,C 180,E1 -7374.016,E2 -7374.016} C_VEL
LIN {X 0,Y 593.146,Z 347.332,A -85,B 0,C 180,E1 -7377.004,E2 -7377.004} C_VEL
LIN {X 0,Y 593.145,Z 347.341,A -85,B 0,C 180,E1 -7380.386,E2 -7380.386} C_VEL
LIN {X 0,Y 593.171,Z 347.333,A -85,B 0,C 180,E1 -7383.382,E2 -7383.382} C_VEL
LIN {X 0,Y 593.139,Z 347.328,A -85,B 0,C 180,E1 -7386.582,E2 -7386.582} C_VEL
LIN {X 0,Y 593.185,Z 347.341,A -85,B 0,C 180,E1 -7389.606,E2 -7389.606} C_VEL
LIN {X 0,Y 593.141,Z 347.344,A -85,B 0,C 180,E1 -7392.758,E2 -7392.758} C_VEL
LIN {X 0,Y 593.19,Z 347.326,A -85,B 0,C 180,E1 -7395.747,E2 -7395.747} C_VEL
LIN {X 0,Y 593.14,Z 347.339,A -85,B 0,C 180,E1 -7398.885,E2 -7398.885} C_VEL
LIN {X 0,Y 593.203,Z 347.338,A -85,B 0,C 180,E1 -7402.018,E2 -7402.018} C_VEL
LIN {X 0,Y 593.139,Z 347.342,A -85,B 0,C 180,E1 -7405.143,E2 -7405.143} C_VEL
LIN {X 0,Y 593.201,Z 347.328,A -85,B 0,C 180,E1 -7408.272,E2 -7408.272} C_VEL
LIN {X 0,Y 593.138,Z 347.331,A -85,B 0,C 180,E1 -7411.28,E2 -7411.28} C_VEL
LIN {X 0,Y 593.198,Z 347.33,A -85,B 0,C 180,E1 -7414.38,E2 -7414.38} C_VEL
LIN {X 0,Y 593.14,Z 347.333,A -85,B 0,C 180,E1 -7417.486,E2 -7417.486} C_VEL
LIN {X 0,Y 593.188,Z 347.333,A -85,B 0,C 180,E1 -7420.665,E2 -7420.665} C_VEL
LIN {X 0,Y 593.149,Z 347.346,A -85,B 0,C 180,E1 -7423.722,E2 -7423.722} C_VEL
LIN {X 0,Y 593.164,Z 347.47,A -85,B 0,C 180,E1 -7425.724,E2 -7425.724} C_VEL
LIN {X 0,Y 594.718,Z 351.141,A -85,B 0,C 180,E1 -7426.247,E2 -7426.247} C_VEL
LIN {X 0,Y 609.826,Z 374.57,A -85,B 0,C 180,E1 -7427.967,E2 -7427.967} C_VEL
LIN {X 0,Y 621.376,Z 393.411,A -85,B 0,C 180,E1 -7429.21,E2 -7429.21} C_VEL
LIN {X 0,Y 624.055,Z 398.23,A -85,B 0,C 180,E1 -7429.495,E2 -7429.495} C_VEL
LIN {X 0,Y 621.779,Z 510.962,A -85,B 0,C 180,E1 -7430.981,E2 -7430.981} C_VEL
LIN {X 0,Y 620.836,Z 518.66,A -85,B 0,C 180,E1 -7431.023,E2 -7431.023} C_VEL
LIN {X 0,Y 615.578,Z 539.219,A -85,B 0,C 180,E1 -7430.927,E2 -7430.927} C_VEL
LIN {X 0,Y 614.866,Z 545.822,A -85,B 0,C 180,E1 -7430.97,E2 -7430.97} C_VEL
LIN {X 0,Y 610.87,Z 739.089,A -85,B 0,C 180,E1 -7433.525,E2 -7433.525} C_VEL
LIN {X 0,Y 609.722,Z 764.923,A -85,B 0,C 180,E1 -7434.028,E2 -7434.028} C_VEL
LIN {X 0,Y 608.488,Z 785.135,A -85,B 0,C 180,E1 -7434.558,E2 -7434.558} C_VEL
LIN {X 0,Y 606.898,Z 807.794,A -85,B 0,C 180,E1 -7435.298,E2 -7435.298} C_VEL
LIN {X 0,Y 604.896,Z 830.349,A -85,B 0,C 180,E1 -7436.22,E2 -7436.22} C_VEL
LIN {X 0,Y 603.028,Z 849.958,A -85,B 0,C 180,E1 -7437.166,E2 -7437.166} C_VEL
LIN {X 0,Y 600.674,Z 872.184,A -85,B 0,C 180,E1 -7438.431,E2 -7438.431} C_VEL
LIN {X 0,Y 598.603,Z 890.601,A -85,B 0,C 180,E1 -7439.65,E2 -7439.65} C_VEL
LIN {X 0,Y 596.187,Z 911.336,A -85,B 0,C 180,E1 -7441.227,E2 -7441.227} C_VEL
LIN {X 0,Y 594.073,Z 928.736,A -85,B 0,C 180,E1 -7442.754,E2 -7442.754} C_VEL
LIN {X 0,Y 592.043,Z 946.183,A -85,B 0,C 180,E1 -7444.49,E2 -7444.49} C_VEL
LIN {X 0,Y 590.155,Z 962.156,A -85,B 0,C 180,E1 -7446.325,E2 -7446.325} C_VEL
LIN {X 0,Y 588.473,Z 977.818,A -85,B 0,C 180,E1 -7448.364,E2 -7448.364} C_VEL
LIN {X 0,Y 587.079,Z 991.214,A -85,B 0,C 180,E1 -7450.396,E2 -7450.396} C_VEL
LIN {X 0,Y 586.01,Z 1003.537,A -85,B 0,C 180,E1 -7452.524,E2 -7452.524} C_VEL
LIN {X 0,Y 585.128,Z 1015.176,A -85,B 0,C 180,E1 -7454.906,E2 -7454.906} C_VEL
LIN {X 0,Y 584.581,Z 1024.607,A -85,B 0,C 180,E1 -7457.153,E2 -7457.153} C_VEL
LIN {X 0,Y 584.224,Z 1032.375,A -85,B 0,C 180,E1 -7459.448,E2 -7459.448} C_VEL
LIN {X 0,Y 584.041,Z 1038.139,A -85,B 0,C 180,E1 -7461.533,E2 -7461.533} C_VEL
LIN {X 0,Y 583.949,Z 1043.26,A -85,B 0,C 180,E1 -7464.005,E2 -7464.005} C_VEL
LIN {X 0,Y 583.917,Z 1046.182,A -85,B 0,C 180,E1 -7466.073,E2 -7466.073} C_VEL
LIN {X 0,Y 583.896,Z 1048.13,A -85,B 0,C 180,E1 -7468.43,E2 -7468.43} C_VEL
LIN {X 0,Y 583.897,Z 1048.359,A -85,B 0,C 180,E1 -7470.687,E2 -7470.687} C_VEL
LIN {X 0,Y 583.902,Z 1047.389,A -85,B 0,C 180,E1 -7472.748,E2 -7472.748} C_VEL
LIN {X 0,Y 583.925,Z 1044.684,A -85,B 0,C 180,E1 -7475.207,E2 -7475.207} C_VEL
LIN {X 0,Y 583.978,Z 1040.783,A -85,B 0,C 180,E1 -7477.378,E2 -7477.378} C_VEL
LIN {X 0,Y 584.126,Z 1035.454,A -85,B 0,C 180,E1 -7479.604,E2 -7479.604} C_VEL
LIN {X 0,Y 584.402,Z 1028.113,A -85,B 0,C 180,E1 -7481.948,E2 -7481.948} C_VEL
LIN {X 0,Y 584.791,Z 1020.521,A -85,B 0,C 180,E1 -7483.951,E2 -7483.951} C_VEL
LIN {X 0,Y 585.515,Z 1009.6,A -85,B 0,C 180,E1 -7486.366,E2 -7486.366} C_VEL
LIN {X 0,Y 586.376,Z 998.933,A -85,B 0,C 180,E1 -7488.389,E2 -7488.389} C_VEL
LIN {X 0,Y 587.617,Z 986.028,A -85,B 0,C 180,E1 -7490.52,E2 -7490.52} C_VEL
LIN {X 0,Y 589.014,Z 972.413,A -85,B 0,C 180,E1 -7492.455,E2 -7492.455} C_VEL
LIN {X 0,Y 590.807,Z 956.751,A -85,B 0,C 180,E1 -7494.422,E2 -7494.422} C_VEL
LIN {X 0,Y 592.73,Z 940.054,A -85,B 0,C 180,E1 -7496.23,E2 -7496.23} C_VEL
LIN {X 0,Y 594.906,Z 922.245,A -85,B 0,C 180,E1 -7497.935,E2 -7497.935} C_VEL
LIN {X 0,Y 597.138,Z 903.068,A -85,B 0,C 180,E1 -7499.519,E2 -7499.519} C_VEL
LIN {X 0,Y 599.31,Z 884.496,A -85,B 0,C 180,E1 -7500.866,E2 -7500.866} C_VEL
LIN {X 0,Y 601.739,Z 862.471,A -85,B 0,C 180,E1 -7502.235,E2 -7502.235} C_VEL
LIN {X 0,Y 603.657,Z 843.548,A -85,B 0,C 180,E1 -7503.248,E2 -7503.248} C_VEL
LIN {X 0,Y 605.832,Z 820.182,A -85,B 0,C 180,E1 -7504.307,E2 -7504.307} C_VEL
LIN {X 0,Y 607.476,Z 799.18,A -85,B 0,C 180,E1 -7505.091,E2 -7505.091} C_VEL
LIN {X 0,Y 609.14,Z 775.338,A -85,B 0,C 180,E1 -7505.812,E2 -7505.812} C_VEL
LIN {X 0,Y 610.35,Z 752.179,A -85,B 0,C 180,E1 -7506.333,E2 -7506.333} C_VEL
LIN {X 0,Y 611.214,Z 728.402,A -85,B 0,C 180,E1 -7506.725,E2 -7506.725} C_VEL
LIN {X 0,Y 616.399,Z 474.236,A -85,B 0,C 180,E1 -7510.067,E2 -7510.067} C_VEL
LIN {X 0,Y 617.783,Z 400.898,A -85,B 0,C 180,E1 -7511.059,E2 -7511.059} C_VEL
LIN {X 0,Y 605.4,Z 380.52,A -85,B 0,C 180,E1 -7512.415,E2 -7512.415} C_VEL
LIN {X 0,Y 595.632,Z 365.36,A -85,B 0,C 180,E1 -7513.532,E2 -7513.532} C_VEL
LIN {X 0,Y 589.176,Z 355.763,A -85,B 0,C 180,E1 -7514.295,E2 -7514.295} C_VEL
LIN {X 0,Y 586.003,Z 350.942,A -85,B 0,C 180,E1 -7514.71,E2 -7514.71} C_VEL
LIN {X 0,Y 585.22,Z 348.305,A -85,B 0,C 180,E1 -7515.118,E2 -7515.118} C_VEL
LIN {X 0,Y 585.197,Z 348.29,A -85,B 0,C 180,E1 -7518.343,E2 -7518.343} C_VEL
LIN {X 0,Y 585.236,Z 348.334,A -85,B 0,C 180,E1 -7521.334,E2 -7521.334} C_VEL
LIN {X 0,Y 585.197,Z 348.335,A -85,B 0,C 180,E1 -7524.59,E2 -7524.59} C_VEL
LIN {X 0,Y 585.26,Z 348.326,A -85,B 0,C 180,E1 -7527.745,E2 -7527.745} C_VEL
LIN {X 0,Y 585.195,Z 348.335,A -85,B 0,C 180,E1 -7530.859,E2 -7530.859} C_VEL
LIN {X 0,Y 585.257,Z 348.331,A -85,B 0,C 180,E1 -7533.981,E2 -7533.981} C_VEL
LIN {X 0,Y 585.196,Z 348.324,A -85,B 0,C 180,E1 -7537.072,E2 -7537.072} C_VEL
LIN {X 0,Y 585.237,Z 348.315,A -85,B 0,C 180,E1 -7540.287,E2 -7540.287} C_VEL
LIN {X 0,Y 585.201,Z 348.334,A -85,B 0,C 180,E1 -7543.319,E2 -7543.319} C_VEL
LIN {X 0,Y 585.212,Z 348.332,A -85,B 0,C 180,E1 -7546.664,E2 -7546.664} C_VEL
LIN {X 0,Y 585.216,Z 348.316,A -85,B 0,C 180,E1 -7549.665,E2 -7549.665} C_VEL
LIN {X 0,Y 585.198,Z 348.323,A -85,B 0,C 180,E1 -7552.933,E2 -7552.933} C_VEL
LIN {X 0,Y 585.24,Z 348.333,A -85,B 0,C 180,E1 -7555.983,E2 -7555.983} C_VEL
LIN {X 0,Y 585.194,Z 348.323,A -85,B 0,C 180,E1 -7559.217,E2 -7559.217} C_VEL
LIN {X 0,Y 585.253,Z 348.315,A -85,B 0,C 180,E1 -7562.252,E2 -7562.252} C_VEL
LIN {X 0,Y 585.194,Z 348.333,A -85,B 0,C 180,E1 -7565.392,E2 -7565.392} C_VEL
LIN {X 0,Y 585.258,Z 348.318,A -85,B 0,C 180,E1 -7568.548,E2 -7568.548} C_VEL
LIN {X 0,Y 585.193,Z 348.327,A -85,B 0,C 180,E1 -7571.632,E2 -7571.632} C_VEL
LIN {X 0,Y 585.242,Z 348.327,A -85,B 0,C 180,E1 -7574.849,E2 -7574.849} C_VEL
LIN {X 0,Y 585.199,Z 348.327,A -85,B 0,C 180,E1 -7577.912,E2 -7577.912} C_VEL
LIN {X 0,Y 585.21,Z 348.323,A -85,B 0,C 180,E1 -7581.237,E2 -7581.237} C_VEL
LIN {X 0,Y 585.211,Z 348.323,A -85,B 0,C 180,E1 -7584.162,E2 -7584.162} C_VEL
LIN {X 0,Y 585.202,Z 348.325,A -85,B 0,C 180,E1 -7587.473,E2 -7587.473} C_VEL
LIN {X 0,Y 585.22,Z 348.332,A -85,B 0,C 180,E1 -7590.38,E2 -7590.38} C_VEL
LIN {X 0,Y 585.2,Z 348.332,A -85,B 0,C 180,E1 -7593.614,E2 -7593.614} C_VEL
LIN {X 0,Y 585.247,Z 348.323,A -85,B 0,C 180,E1 -7596.747,E2 -7596.747} C_VEL
LIN {X 0,Y 585.19,Z 348.305,A -85,B 0,C 180,E1 -7599.898,E2 -7599.898} C_VEL
LIN {X 0,Y 585.252,Z 348.434,A -85,B 0,C 180,E1 -7602.769,E2 -7602.769} C_VEL
LIN {X 0,Y 592.86,Z 366.937,A -85,B 0,C 180,E1 -7605.376,E2 -7605.376} C_VEL
LIN {X 0,Y 595.802,Z 374.005,A -85,B 0,C 180,E1 -7606.294,E2 -7606.294} C_VEL
LIN {X 0,Y 609.663,Z 396.837,A -85,B 0,C 180,E1 -7607.875,E2 -7607.875} C_VEL
LIN {X 0,Y 616.005,Z 408.091,A -85,B 0,C 180,E1 -7608.574,E2 -7608.574} C_VEL
LIN {X 0,Y 617.872,Z 417.427,A -85,B 0,C 180,E1 -7608.867,E2 -7608.867} C_VEL
LIN {X 0,Y 612.43,Z 681.543,A -85,B 0,C 180,E1 -7612.353,E2 -7612.353} C_VEL
LIN {X 0,Y 610.619,Z 766.58,A -85,B 0,C 180,E1 -7613.484,E2 -7613.484} C_VEL
LIN {X 0,Y 609.39,Z 791.992,A -85,B 0,C 180,E1 -7613.98,E2 -7613.98} C_VEL
LIN {X 0,Y 608.043,Z 813.209,A -85,B 0,C 180,E1 -7614.537,E2 -7614.537} C_VEL
LIN {X 0,Y 606.23,Z 837.562,A -85,B 0,C 180,E1 -7615.349,E2 -7615.349} C_VEL
LIN {X 0,Y 604.443,Z 857.737,A -85,B 0,C 180,E1 -7616.175,E2 -7616.175} C_VEL
LIN {X 0,Y 602.534,Z 877.777,A -85,B 0,C 180,E1 -7617.136,E2 -7617.136} C_VEL
LIN {X 0,Y 600.18,Z 900.134,A -85,B 0,C 180,E1 -7618.402,E2 -7618.402} C_VEL
LIN {X 0,Y 598.175,Z 918.449,A -85,B 0,C 180,E1 -7619.602,E2 -7619.602} C_VEL
LIN {X 0,Y 595.699,Z 940.329,A -85,B 0,C 180,E1 -7621.256,E2 -7621.256} C_VEL
LIN {X 0,Y 593.722,Z 957.373,A -85,B 0,C 180,E1 -7622.737,E2 -7622.737} C_VEL
LIN {X 0,Y 591.637,Z 976.013,A -85,B 0,C 180,E1 -7624.579,E2 -7624.579} C_VEL
LIN {X 0,Y 589.938,Z 991.354,A -85,B 0,C 180,E1 -7626.316,E2 -7626.316} C_VEL
LIN {X 0,Y 588.4,Z 1006.591,A -85,B 0,C 180,E1 -7628.256,E2 -7628.256} C_VEL
LIN {X 0,Y 587.052,Z 1020.359,A -85,B 0,C 180,E1 -7630.291,E2 -7630.291} C_VEL
LIN {X 0,Y 586.054,Z 1032.454,A -85,B 0,C 180,E1 -7632.32,E2 -7632.32} C_VEL
LIN {X 0,Y 585.221,Z 1043.718,A -85,B 0,C 180,E1 -7634.542,E2 -7634.542} C_VEL
LIN {X 0,Y 584.69,Z 1052.366,A -85,B 0,C 180,E1 -7636.551,E2 -7636.551} C_VEL
LIN {X 0,Y 584.278,Z 1060.997,A -85,B 0,C 180,E1 -7638.95,E2 -7638.95} C_VEL
LIN {X 0,Y 584.055,Z 1067.008,A -85,B 0,C 180,E1 -7641.047,E2 -7641.047} C_VEL
LIN {X 0,Y 583.953,Z 1071.928,A -85,B 0,C 180,E1 -7643.215,E2 -7643.215} C_VEL
LIN {X 0,Y 583.915,Z 1075.667,A -85,B 0,C 180,E1 -7645.58,E2 -7645.58} C_VEL
LIN {X 0,Y 583.91,Z 1077.63,A -85,B 0,C 180,E1 -7647.645,E2 -7647.645} C_VEL
LIN {X 0,Y 583.916,Z 1078.5,A -85,B 0,C 180,E1 -7650,E2 -7650} C_VEL
LIN {X 0,Y 583.91,Z 1077.63,A -85,B 0,C 180,E1 -7652.355,E2 -7652.355} C_VEL
LIN {X 0,Y 583.915,Z 1075.666,A -85,B 0,C 180,E1 -7654.419,E2 -7654.419} C_VEL
LIN {X 0,Y 583.961,Z 1071.721,A -85,B 0,C 180,E1 -7656.884,E2 -7656.884} C_VEL
LIN {X 0,Y 584.056,Z 1066.983,A -85,B 0,C 180,E1 -7658.963,E2 -7658.963} C_VEL
LIN {X 0,Y 584.29,Z 1060.693,A -85,B 0,C 180,E1 -7661.15,E2 -7661.15} C_VEL
LIN {X 0,Y 584.69,Z 1052.365,A -85,B 0,C 180,E1 -7663.449,E2 -7663.449} C_VEL
LIN {X 0,Y 585.236,Z 1043.516,A -85,B 0,C 180,E1 -7665.503,E2 -7665.503} C_VEL
LIN {X 0,Y 586.099,Z 1031.88,A -85,B 0,C 180,E1 -7667.781,E2 -7667.781} C_VEL
LIN {X 0,Y 587.052,Z 1020.363,A -85,B 0,C 180,E1 -7669.709,E2 -7669.709} C_VEL
LIN {X 0,Y 588.469,Z 1005.819,A -85,B 0,C 180,E1 -7671.846,E2 -7671.846} C_VEL
LIN {X 0,Y 590.032,Z 990.502,A -85,B 0,C 180,E1 -7673.786,E2 -7673.786} C_VEL
LIN {X 0,Y 591.925,Z 973.565,A -85,B 0,C 180,E1 -7675.684,E2 -7675.684} C_VEL
LIN {X 0,Y 593.92,Z 955.695,A -85,B 0,C 180,E1 -7677.416,E2 -7677.416} C_VEL
LIN {X 0,Y 596.153,Z 936.638,A -85,B 0,C 180,E1 -7679.049,E2 -7679.049} C_VEL
LIN {X 0,Y 598.376,Z 916.532,A -85,B 0,C 180,E1 -7680.53,E2 -7680.53} C_VEL
LIN {X 0,Y 600.659,Z 896.052,A -85,B 0,C 180,E1 -7681.85,E2 -7681.85} C_VEL
LIN {X 0,Y 602.822,Z 874.753,A -85,B 0,C 180,E1 -7683.016,E2 -7683.016} C_VEL
LIN {X 0,Y 604.643,Z 855.633,A -85,B 0,C 180,E1 -7683.917,E2 -7683.917} C_VEL
LIN {X 0,Y 606.657,Z 832.072,A -85,B 0,C 180,E1 -7684.853,E2 -7684.853} C_VEL
LIN {X 0,Y 608.247,Z 809.891,A -85,B 0,C 180,E1 -7685.559,E2 -7685.559} C_VEL
LIN {X 0,Y 609.76,Z 785.674,A -85,B 0,C 180,E1 -7686.166,E2 -7686.166} C_VEL
LIN {X 0,Y 610.776,Z 761.607,A -85,B 0,C 180,E1 -7686.589,E2 -7686.589} C_VEL
LIN {X 0,Y 615.522,Z 526.574,A -85,B 0,C 180,E1 -7689.685,E2 -7689.685} C_VEL
LIN {X 0,Y 617.706,Z 415.808,A -85,B 0,C 180,E1 -7691.168,E2 -7691.168} C_VEL
LIN {X 0,Y 615.561,Z 407.003,A -85,B 0,C 180,E1 -7691.476,E2 -7691.476} C_VEL
LIN {X 0,Y 601.951,Z 384.02,A -85,B 0,C 180,E1 -7692.987,E2 -7692.987} C_VEL
LIN {X 0,Y 595.407,Z 373.18,A -85,B 0,C 180,E1 -7693.78,E2 -7693.78} C_VEL
LIN {X 0,Y 588.271,Z 355.831,A -85,B 0,C 180,E1 -7696.161,E2 -7696.161} C_VEL
LIN {X 0,Y 585.239,Z 348.328,A -85,B 0,C 180,E1 -7697.26,E2 -7697.26} C_VEL
LIN {X 0,Y 585.201,Z 348.324,A -85,B 0,C 180,E1 -7700.28,E2 -7700.28} C_VEL
LIN {X 0,Y 585.21,Z 348.283,A -85,B 0,C 180,E1 -7703.586,E2 -7703.586} C_VEL
LIN {X 0,Y 585.221,Z 348.322,A -85,B 0,C 180,E1 -7706.667,E2 -7706.667} C_VEL
LIN {X 0,Y 585.2,Z 348.332,A -85,B 0,C 180,E1 -7709.958,E2 -7709.958} C_VEL
LIN {X 0,Y 585.241,Z 348.316,A -85,B 0,C 180,E1 -7712.969,E2 -7712.969} C_VEL
LIN {X 0,Y 585.198,Z 348.322,A -85,B 0,C 180,E1 -7716.112,E2 -7716.112} C_VEL
LIN {X 0,Y 585.252,Z 348.321,A -85,B 0,C 180,E1 -7719.153,E2 -7719.153} C_VEL
LIN {X 0,Y 585.197,Z 348.332,A -85,B 0,C 180,E1 -7722.294,E2 -7722.294} C_VEL
LIN {X 0,Y 585.266,Z 348.323,A -85,B 0,C 180,E1 -7725.455,E2 -7725.455} C_VEL
LIN {X 0,Y 585.195,Z 348.32,A -85,B 0,C 180,E1 -7728.568,E2 -7728.568} C_VEL
LIN {X 0,Y 585.253,Z 348.318,A -85,B 0,C 180,E1 -7731.749,E2 -7731.749} C_VEL
LIN {X 0,Y 585.2,Z 348.332,A -85,B 0,C 180,E1 -7734.804,E2 -7734.804} C_VEL
LIN {X 0,Y 585.231,Z 348.319,A -85,B 0,C 180,E1 -7738.042,E2 -7738.042} C_VEL
LIN {X 0,Y 585.202,Z 348.327,A -85,B 0,C 180,E1 -7740.979,E2 -7740.979} C_VEL
LIN {X 0,Y 585.218,Z 348.334,A -85,B 0,C 180,E1 -7744.311,E2 -7744.311} C_VEL
LIN {X 0,Y 585.223,Z 348.314,A -85,B 0,C 180,E1 -7747.362,E2 -7747.362} C_VEL
LIN {X 0,Y 585.203,Z 348.32,A -85,B 0,C 180,E1 -7750.634,E2 -7750.634} C_VEL
LIN {X 0,Y 585.253,Z 348.329,A -85,B 0,C 180,E1 -7753.738,E2 -7753.738} C_VEL
LIN {X 0,Y 585.201,Z 348.331,A -85,B 0,C 180,E1 -7756.897,E2 -7756.897} C_VEL
LIN {X 0,Y 585.262,Z 348.314,A -85,B 0,C 180,E1 -7760.084,E2 -7760.084} C_VEL
LIN {X 0,Y 585.201,Z 348.327,A -85,B 0,C 180,E1 -7763.185,E2 -7763.185} C_VEL
LIN {X 0,Y 585.25,Z 348.33,A -85,B 0,C 180,E1 -7766.373,E2 -7766.373} C_VEL
LIN {X 0,Y 585.208,Z 348.332,A -85,B 0,C 180,E1 -7769.477,E2 -7769.477} C_VEL
LIN {X 0,Y 585.223,Z 348.335,A -85,B 0,C 180,E1 -7772.795,E2 -7772.795} C_VEL
LIN {X 0,Y 585.23,Z 348.329,A -85,B 0,C 180,E1 -7775.876,E2 -7775.876} C_VEL
LIN {X 0,Y 585.209,Z 348.334,A -85,B 0,C 180,E1 -7779.131,E2 -7779.131} C_VEL
LIN {X 0,Y 585.25,Z 348.328,A -85,B 0,C 180,E1 -7782.178,E2 -7782.178} C_VEL
LIN {X 0,Y 585.235,Z 348.445,A -85,B 0,C 180,E1 -7785.037,E2 -7785.037} C_VEL
LIN {X 0,Y 586.447,Z 351.722,A -85,B 0,C 180,E1 -7785.472,E2 -7785.472} C_VEL
LIN {X 0,Y 594.153,Z 363.118,A -85,B 0,C 180,E1 -7786.391,E2 -7786.391} C_VEL
LIN {X 0,Y 604.801,Z 379.564,A -85,B 0,C 180,E1 -7787.612,E2 -7787.612} C_VEL
LIN {X 0,Y 616.684,Z 399.091,A -85,B 0,C 180,E1 -7788.916,E2 -7788.916} C_VEL
LIN {X 0,Y 617.925,Z 401.521,A -85,B 0,C 180,E1 -7789.054,E2 -7789.054} C_VEL
LIN {X 0,Y 614.866,Z 545.822,A -85,B 0,C 180,E1 -7790.97,E2 -7790.97} C_VEL
LIN {X 0,Y 613.948,Z 553.517,A -85,B 0,C 180,E1 -7791.014,E2 -7791.014} C_VEL
LIN {X 0,Y 608.682,Z 574.074,A -85,B 0,C 180,E1 -7790.916,E2 -7790.916} C_VEL
LIN {X 0,Y 607.927,Z 580.681,A -85,B 0,C 180,E1 -7790.957,E2 -7790.957} C_VEL
LIN {X 0,Y 604.45,Z 739.439,A -85,B 0,C 180,E1 -7793.075,E2 -7793.075} C_VEL
LIN {X 0,Y 603.244,Z 765.285,A -85,B 0,C 180,E1 -7793.584,E2 -7793.584} C_VEL
LIN {X 0,Y 601.939,Z 785.701,A -85,B 0,C 180,E1 -7794.124,E2 -7794.124} C_VEL
LIN {X 0,Y 600.263,Z 808.375,A -85,B 0,C 180,E1 -7794.874,E2 -7794.874} C_VEL
LIN {X 0,Y 598.235,Z 830.26,A -85,B 0,C 180,E1 -7795.776,E2 -7795.776} C_VEL
LIN {X 0,Y 596.239,Z 850.184,A -85,B 0,C 180,E1 -7796.744,E2 -7796.744} C_VEL
LIN {X 0,Y 593.743,Z 872.549,A -85,B 0,C 180,E1 -7798.029,E2 -7798.029} C_VEL
LIN {X 0,Y 591.575,Z 890.828,A -85,B 0,C 180,E1 -7799.25,E2 -7799.25} C_VEL
LIN {X 0,Y 589.032,Z 911.562,A -85,B 0,C 180,E1 -7800.844,E2 -7800.844} C_VEL
LIN {X 0,Y 586.808,Z 928.896,A -85,B 0,C 180,E1 -7802.382,E2 -7802.382} C_VEL
LIN {X 0,Y 584.64,Z 946.408,A -85,B 0,C 180,E1 -7804.144,E2 -7804.144} C_VEL
LIN {X 0,Y 582.636,Z 962.381,A -85,B 0,C 180,E1 -7806.001,E2 -7806.001} C_VEL
LIN {X 0,Y 580.836,Z 978.042,A -85,B 0,C 180,E1 -7808.065,E2 -7808.065} C_VEL
LIN {X 0,Y 579.328,Z 991.665,A -85,B 0,C 180,E1 -7810.161,E2 -7810.161} C_VEL
LIN {X 0,Y 578.175,Z 1004.108,A -85,B 0,C 180,E1 -7812.345,E2 -7812.345} C_VEL
LIN {X 0,Y 577.261,Z 1015.052,A -85,B 0,C 180,E1 -7814.632,E2 -7814.632} C_VEL
LIN {X 0,Y 576.66,Z 1024.233,A -85,B 0,C 180,E1 -7816.871,E2 -7816.871} C_VEL
LIN {X 0,Y 576.251,Z 1032.376,A -85,B 0,C 180,E1 -7819.3,E2 -7819.3} C_VEL
LIN {X 0,Y 576.047,Z 1038.141,A -85,B 0,C 180,E1 -7821.415,E2 -7821.415} C_VEL
LIN {X 0,Y 575.953,Z 1043.261,A -85,B 0,C 180,E1 -7823.921,E2 -7823.921} C_VEL
LIN {X 0,Y 575.918,Z 1046.182,A -85,B 0,C 180,E1 -7826.018,E2 -7826.018} C_VEL
LIN {X 0,Y 575.896,Z 1048.131,A -85,B 0,C 180,E1 -7828.408,E2 -7828.408} C_VEL
LIN {X 0,Y 575.898,Z 1048.358,A -85,B 0,C 180,E1 -7830.696,E2 -7830.696} C_VEL
LIN {X 0,Y 575.902,Z 1047.456,A -85,B 0,C 180,E1 -7832.687,E2 -7832.687} C_VEL
LIN {X 0,Y 575.926,Z 1045.002,A -85,B 0,C 180,E1 -7835.08,E2 -7835.08} C_VEL
LIN {X 0,Y 575.98,Z 1040.988,A -85,B 0,C 180,E1 -7837.381,E2 -7837.381} C_VEL
LIN {X 0,Y 576.124,Z 1036.079,A -85,B 0,C 180,E1 -7839.49,E2 -7839.49} C_VEL
LIN {X 0,Y 576.428,Z 1028.463,A -85,B 0,C 180,E1 -7842.014,E2 -7842.014} C_VEL
LIN {X 0,Y 576.897,Z 1020.194,A -85,B 0,C 180,E1 -7844.248,E2 -7844.248} C_VEL
LIN {X 0,Y 577.709,Z 1009.307,A -85,B 0,C 180,E1 -7846.697,E2 -7846.697} C_VEL
LIN {X 0,Y 578.595,Z 999.149,A -85,B 0,C 180,E1 -7848.645,E2 -7848.645} C_VEL
LIN {X 0,Y 579.956,Z 985.875,A -85,B 0,C 180,E1 -7850.86,E2 -7850.86} C_VEL
LIN {X 0,Y 581.481,Z 972.171,A -85,B 0,C 180,E1 -7852.826,E2 -7852.826} C_VEL
LIN {X 0,Y 583.399,Z 956.331,A -85,B 0,C 180,E1 -7854.829,E2 -7854.829} C_VEL
LIN {X 0,Y 585.442,Z 939.764,A -85,B 0,C 180,E1 -7856.637,E2 -7856.637} C_VEL
LIN {X 0,Y 587.712,Z 922.157,A -85,B 0,C 180,E1 -7858.338,E2 -7858.338} C_VEL
LIN {X 0,Y 590.073,Z 902.95,A -85,B 0,C 180,E1 -7859.936,E2 -7859.936} C_VEL
LIN {X 0,Y 592.431,Z 883.975,A -85,B 0,C 180,E1 -7861.321,E2 -7861.321} C_VEL
LIN {X 0,Y 594.885,Z 862.678,A -85,B 0,C 180,E1 -7862.652,E2 -7862.652} C_VEL
LIN {X 0,Y 596.897,Z 843.755,A -85,B 0,C 180,E1 -7863.675,E2 -7863.675} C_VEL
LIN {X 0,Y 599.179,Z 820.385,A -85,B 0,C 180,E1 -7864.742,E2 -7864.742} C_VEL
LIN {X 0,Y 600.939,Z 798.957,A -85,B 0,C 180,E1 -7865.547,E2 -7865.547} C_VEL
LIN {X 0,Y 602.707,Z 774.588,A -85,B 0,C 180,E1 -7866.281,E2 -7866.281} C_VEL
LIN {X 0,Y 603.923,Z 752.209,A -85,B 0,C 180,E1 -7866.786,E2 -7866.786} C_VEL
LIN {X 0,Y 604.835,Z 728.071,A -85,B 0,C 180,E1 -7867.186,E2 -7867.186} C_VEL
LIN {X 0,Y 610.303,Z 473.872,A -85,B 0,C 180,E1 -7870.558,E2 -7870.558} C_VEL
LIN {X 0,Y 611.722,Z 404.284,A -85,B 0,C 180,E1 -7871.507,E2 -7871.507} C_VEL
LIN {X 0,Y 598.793,Z 382.833,A -85,B 0,C 180,E1 -7872.961,E2 -7872.961} C_VEL
LIN {X 0,Y 584.923,Z 361.758,A -85,B 0,C 180,E1 -7874.603,E2 -7874.603} C_VEL
LIN {X 0,Y 577.841,Z 351.322,A -85,B 0,C 180,E1 -7875.508,E2 -7875.508} C_VEL
LIN {X 0,Y 577.306,Z 349.312,A -85,B 0,C 180,E1 -7875.811,E2 -7875.811} C_VEL
LIN {X 0,Y 577.256,Z 349.277,A -85,B 0,C 180,E1 -7878.893,E2 -7878.893} C_VEL
LIN {X 0,Y 577.278,Z 349.314,A -85,B 0,C 180,E1 -7882.182,E2 -7882.182} C_VEL
LIN {X 0,Y 577.282,Z 349.314,A -85,B 0,C 180,E1 -7885.26,E2 -7885.26} C_VEL
LIN {X 0,Y 577.26,Z 349.313,A -85,B 0,C 180,E1 -7888.576,E2 -7888.576} C_VEL
LIN {X 0,Y 577.315,Z 349.309,A -85,B 0,C 180,E1 -7891.669,E2 -7891.669} C_VEL
LIN {X 0,Y 577.258,Z 349.322,A -85,B 0,C 180,E1 -7894.779,E2 -7894.779} C_VEL
LIN {X 0,Y 577.331,Z 349.318,A -85,B 0,C 180,E1 -7897.924,E2 -7897.924} C_VEL
LIN {X 0,Y 577.256,Z 349.312,A -85,B 0,C 180,E1 -7901.1,E2 -7901.1} C_VEL
LIN {X 0,Y 577.301,Z 349.301,A -85,B 0,C 180,E1 -7904.324,E2 -7904.324} C_VEL
LIN {X 0,Y 577.259,Z 349.323,A -85,B 0,C 180,E1 -7907.292,E2 -7907.292} C_VEL
LIN {X 0,Y 577.281,Z 349.319,A -85,B 0,C 180,E1 -7910.63,E2 -7910.63} C_VEL
LIN {X 0,Y 577.269,Z 349.306,A -85,B 0,C 180,E1 -7913.635,E2 -7913.635} C_VEL
LIN {X 0,Y 577.266,Z 349.317,A -85,B 0,C 180,E1 -7916.922,E2 -7916.922} C_VEL
LIN {X 0,Y 577.297,Z 349.314,A -85,B 0,C 180,E1 -7920,E2 -7920} C_VEL
LIN {X 0,Y 577.256,Z 349.302,A -85,B 0,C 180,E1 -7923.177,E2 -7923.177} C_VEL
LIN {X 0,Y 577.321,Z 349.311,A -85,B 0,C 180,E1 -7926.364,E2 -7926.364} C_VEL
LIN {X 0,Y 577.254,Z 349.32,A -85,B 0,C 180,E1 -7929.471,E2 -7929.471} C_VEL
LIN {X 0,Y 577.312,Z 349.304,A -85,B 0,C 180,E1 -7932.707,E2 -7932.707} C_VEL
LIN {X 0,Y 577.257,Z 349.317,A -85,B 0,C 180,E1 -7935.78,E2 -7935.78} C_VEL
LIN {X 0,Y 577.289,Z 349.316,A -85,B 0,C 180,E1 -7939.004,E2 -7939.004} C_VEL
LIN {X 0,Y 577.268,Z 349.317,A -85,B 0,C 180,E1 -7942.078,E2 -7942.078} C_VEL
LIN {X 0,Y 577.263,Z 349.319,A -85,B 0,C 180,E1 -7945.44,E2 -7945.44} C_VEL
LIN {X 0,Y 577.305,Z 349.308,A -85,B 0,C 180,E1 -7948.557,E2 -7948.557} C_VEL
LIN {X 0,Y 577.254,Z 349.315,A -85,B 0,C 180,E1 -7951.735,E2 -7951.735} C_VEL
LIN {X 0,Y 577.316,Z 349.311,A -85,B 0,C 180,E1 -7954.858,E2 -7954.858} C_VEL
LIN {X 0,Y 577.255,Z 349.324,A -85,B 0,C 180,E1 -7957.989,E2 -7957.989} C_VEL
LIN {X 0,Y 577.311,Z 349.275,A -85,B 0,C 180,E1 -7961.159,E2 -7961.159} C_VEL
LIN {X 0,Y 577.286,Z 349.542,A -85,B 0,C 180,E1 -7962.057,E2 -7962.057} C_VEL
LIN {X 0,Y 578.498,Z 352.671,A -85,B 0,C 180,E1 -7962.518,E2 -7962.518} C_VEL
LIN {X 0,Y 585.073,Z 368.039,A -85,B 0,C 180,E1 -7964.758,E2 -7964.758} C_VEL
LIN {X 0,Y 587.366,Z 373.708,A -85,B 0,C 180,E1 -7965.502,E2 -7965.502} C_VEL
LIN {X 0,Y 601.334,Z 396.097,A -85,B 0,C 180,E1 -7967.146,E2 -7967.146} C_VEL
LIN {X 0,Y 610.468,Z 412.228,A -85,B 0,C 180,E1 -7968.181,E2 -7968.181} C_VEL
LIN {X 0,Y 611.792,Z 419.291,A -85,B 0,C 180,E1 -7968.399,E2 -7968.399} C_VEL
LIN {X 0,Y 606.065,Z 682.561,A -85,B 0,C 180,E1 -7971.905,E2 -7971.905} C_VEL
LIN {X 0,Y 604.184,Z 766.38,A -85,B 0,C 180,E1 -7973.03,E2 -7973.03} C_VEL
LIN {X 0,Y 602.88,Z 791.9,A -85,B 0,C 180,E1 -7973.532,E2 -7973.532} C_VEL
LIN {X 0,Y 601.454,Z 813.326,A -85,B 0,C 180,E1 -7974.099,E2 -7974.099} C_VEL
LIN {X 0,Y 599.516,Z 837.93,A -85,B 0,C 180,E1 -7974.931,E2 -7974.931} C_VEL
LIN {X 0,Y 597.656,Z 857.951,A -85,B 0,C 180,E1 -7975.76,E2 -7975.76} C_VEL
LIN {X 0,Y 595.588,Z 878.571,A -85,B 0,C 180,E1 -7976.761,E2 -7976.761} C_VEL
LIN {X 0,Y 593.107,Z 900.733,A -85,B 0,C 180,E1 -7978.038,E2 -7978.038} C_VEL
LIN {X 0,Y 590.883,Z 920.018,A -85,B 0,C 180,E1 -7979.323,E2 -7979.323} C_VEL
LIN {X 0,Y 588.39,Z 940.722,A -85,B 0,C 180,E1 -7980.921,E2 -7980.921} C_VEL
LIN {X 0,Y 586.309,Z 957.711,A -85,B 0,C 180,E1 -7982.418,E2 -7982.418} C_VEL
LIN {X 0,Y 584.038,Z 976.726,A -85,B 0,C 180,E1 -7984.333,E2 -7984.333} C_VEL
LIN {X 0,Y 582.255,Z 991.987,A -85,B 0,C 180,E1 -7986.091,E2 -7986.091} C_VEL
LIN {X 0,Y 580.529,Z 1007.948,A -85,B 0,C 180,E1 -7988.182,E2 -7988.182} C_VEL
LIN {X 0,Y 579.21,Z 1020.781,A -85,B 0,C 180,E1 -7990.118,E2 -7990.118} C_VEL
LIN {X 0,Y 578.112,Z 1033.392,A -85,B 0,C 180,E1 -7992.278,E2 -7992.278} C_VEL
LIN {X 0,Y 577.248,Z 1044.492,A -85,B 0,C 180,E1 -7994.529,E2 -7994.529} C_VEL
LIN {X 0,Y 576.688,Z 1053.566,A -85,B 0,C 180,E1 -7996.667,E2 -7996.667} C_VEL
LIN {X 0,Y 576.271,Z 1061.906,A -85,B 0,C 180,E1 -7999.098,E2 -7999.098} C_VEL
LIN {X 0,Y 576.051,Z 1067.745,A -85,B 0,C 180,E1 -8001.214,E2 -8001.214} C_VEL
LIN {X 0,Y 575.949,Z 1073.014,A -85,B 0,C 180,E1 -8003.721,E2 -8003.721} C_VEL
LIN {X 0,Y 575.914,Z 1076.007,A -85,B 0,C 180,E1 -8005.818,E2 -8005.818} C_VEL
LIN {X 0,Y 575.908,Z 1077.834,A -85,B 0,C 180,E1 -8007.91,E2 -8007.91} C_VEL
LIN {X 0,Y 575.895,Z 1078.416,A -85,B 0,C 180,E1 -8010.398,E2 -8010.398} C_VEL
LIN {X 0,Y 575.908,Z 1077.561,A -85,B 0,C 180,E1 -8012.488,E2 -8012.488} C_VEL
LIN {X 0,Y 575.923,Z 1075.438,A -85,B 0,C 180,E1 -8014.68,E2 -8014.68} C_VEL
LIN {X 0,Y 575.989,Z 1071.308,A -85,B 0,C 180,E1 -8017.18,E2 -8017.18} C_VEL
LIN {X 0,Y 576.101,Z 1066.474,A -85,B 0,C 180,E1 -8019.289,E2 -8019.289} C_VEL
LIN {X 0,Y 576.405,Z 1059.011,A -85,B 0,C 180,E1 -8021.812,E2 -8021.812} C_VEL
LIN {X 0,Y 576.802,Z 1051.511,A -85,B 0,C 180,E1 -8023.841,E2 -8023.841} C_VEL
LIN {X 0,Y 577.46,Z 1041.705,A -85,B 0,C 180,E1 -8026.084,E2 -8026.084} C_VEL
LIN {X 0,Y 578.395,Z 1029.78,A -85,B 0,C 180,E1 -8028.363,E2 -8028.363} C_VEL
LIN {X 0,Y 579.546,Z 1017.571,A -85,B 0,C 180,E1 -8030.396,E2 -8030.396} C_VEL
LIN {X 0,Y 581.09,Z 1002.481,A -85,B 0,C 180,E1 -8032.564,E2 -8032.564} C_VEL
LIN {X 0,Y 582.652,Z 988.572,A -85,B 0,C 180,E1 -8034.322,E2 -8034.322} C_VEL
LIN {X 0,Y 584.845,Z 969.839,A -85,B 0,C 180,E1 -8036.392,E2 -8036.392} C_VEL
LIN {X 0,Y 586.869,Z 953.234,A -85,B 0,C 180,E1 -8037.995,E2 -8037.995} C_VEL
LIN {X 0,Y 589.38,Z 932.391,A -85,B 0,C 180,E1 -8039.751,E2 -8039.751} C_VEL
LIN {X 0,Y 591.586,Z 913.956,A -85,B 0,C 180,E1 -8041.098,E2 -8041.098} C_VEL
LIN {X 0,Y 594.217,Z 891.166,A -85,B 0,C 180,E1 -8042.538,E2 -8042.538} C_VEL
LIN {X 0,Y 596.286,Z 871.5,A -85,B 0,C 180,E1 -8043.598,E2 -8043.598} C_VEL
LIN {X 0,Y 598.49,Z 849.526,A -85,B 0,C 180,E1 -8044.613,E2 -8044.613} C_VEL
LIN {X 0,Y 600.404,Z 826.633,A -85,B 0,C 180,E1 -8045.475,E2 -8045.475} C_VEL
LIN {X 0,Y 602.188,Z 803.366,A -85,B 0,C 180,E1 -8046.186,E2 -8046.186} C_VEL
LIN {X 0,Y 603.578,Z 779.59,A -85,B 0,C 180,E1 -8046.729,E2 -8046.729} C_VEL
LIN {X 0,Y 604.468,Z 757.73,A -85,B 0,C 180,E1 -8047.098,E2 -8047.098} C_VEL
LIN {X 0,Y 609.671,Z 512.441,A -85,B 0,C 180,E1 -8050.352,E2 -8050.352} C_VEL
LIN {X 0,Y 611.63,Z 417.648,A -85,B 0,C 180,E1 -8051.636,E2 -8051.636} C_VEL
LIN {X 0,Y 609.987,Z 411.04,A -85,B 0,C 180,E1 -8051.874,E2 -8051.874} C_VEL
LIN {X 0,Y 596.874,Z 388.933,A -85,B 0,C 180,E1 -8053.361,E2 -8053.361} C_VEL
LIN {X 0,Y 587.044,Z 373.117,A -85,B 0,C 180,E1 -8054.542,E2 -8054.542} C_VEL
LIN {X 0,Y 581.547,Z 359.85,A -85,B 0,C 180,E1 -8056.412,E2 -8056.412} C_VEL
LIN {X 0,Y 578.47,Z 352.63,A -85,B 0,C 180,E1 -8057.48,E2 -8057.48} C_VEL
LIN {X 0,Y 577.254,Z 349.317,A -85,B 0,C 180,E1 -8057.995,E2 -8057.995} C_VEL
LIN {X 0,Y 577.328,Z 349.31,A -85,B 0,C 180,E1 -8061.046,E2 -8061.046} C_VEL
LIN {X 0,Y 577.249,Z 349.267,A -85,B 0,C 180,E1 -8064.163,E2 -8064.163} C_VEL
LIN {X 0,Y 577.303,Z 349.317,A -85,B 0,C 180,E1 -8067.408,E2 -8067.408} C_VEL
LIN {X 0,Y 577.261,Z 349.319,A -85,B 0,C 180,E1 -8070.419,E2 -8070.419} C_VEL
LIN {X 0,Y 577.286,Z 349.321,A -85,B 0,C 180,E1 -8073.678,E2 -8073.678} C_VEL
LIN {X 0,Y 577.276,Z 349.312,A -85,B 0,C 180,E1 -8076.739,E2 -8076.739} C_VEL
LIN {X 0,Y 577.265,Z 349.31,A -85,B 0,C 180,E1 -8080.048,E2 -8080.048} C_VEL
LIN {X 0,Y 577.298,Z 349.313,A -85,B 0,C 180,E1 -8083.083,E2 -8083.083} C_VEL
LIN {X 0,Y 577.26,Z 349.322,A -85,B 0,C 180,E1 -8086.273,E2 -8086.273} C_VEL
LIN {X 0,Y 577.316,Z 349.307,A -85,B 0,C 180,E1 -8089.421,E2 -8089.421} C_VEL
LIN {X 0,Y 577.256,Z 349.303,A -85,B 0,C 180,E1 -8092.536,E2 -8092.536} C_VEL
LIN {X 0,Y 577.316,Z 349.317,A -85,B 0,C 180,E1 -8095.729,E2 -8095.729} C_VEL
LIN {X 0,Y 577.262,Z 349.318,A -85,B 0,C 180,E1 -8098.908,E2 -8098.908} C_VEL
LIN {X 0,Y 577.284,Z 349.305,A -85,B 0,C 180,E1 -8102.184,E2 -8102.184} C_VEL
LIN {X 0,Y 577.28,Z 349.319,A -85,B 0,C 180,E1 -8105.267,E2 -8105.267} C_VEL
LIN {X 0,Y 577.267,Z 349.323,A -85,B 0,C 180,E1 -8108.567,E2 -8108.567} C_VEL
LIN {X 0,Y 577.307,Z 349.3,A -85,B 0,C 180,E1 -8111.692,E2 -8111.692} C_VEL
LIN {X 0,Y 577.261,Z 349.313,A -85,B 0,C 180,E1 -8114.867,E2 -8114.867} C_VEL
LIN {X 0,Y 577.322,Z 349.319,A -85,B 0,C 180,E1 -8118.06,E2 -8118.06} C_VEL
LIN {X 0,Y 577.265,Z 349.318,A -85,B 0,C 180,E1 -8121.224,E2 -8121.224} C_VEL
LIN {X 0,Y 577.299,Z 349.308,A -85,B 0,C 180,E1 -8124.453,E2 -8124.453} C_VEL
LIN {X 0,Y 577.274,Z 349.31,A -85,B 0,C 180,E1 -8127.547,E2 -8127.547} C_VEL
LIN {X 0,Y 577.275,Z 349.309,A -85,B 0,C 180,E1 -8130.844,E2 -8130.844} C_VEL
LIN {X 0,Y 577.302,Z 349.313,A -85,B 0,C 180,E1 -8133.939,E2 -8133.939} C_VEL
LIN {X 0,Y 577.263,Z 349.312,A -85,B 0,C 180,E1 -8137.194,E2 -8137.194} C_VEL
LIN {X 0,Y 577.326,Z 349.307,A -85,B 0,C 180,E1 -8140.372,E2 -8140.372} C_VEL
LIN {X 0,Y 577.266,Z 349.321,A -85,B 0,C 180,E1 -8143.581,E2 -8143.581} C_VEL
LIN {X 0,Y 577.344,Z 349.505,A -85,B 0,C 180,E1 -8144.335,E2 -8144.335} C_VEL
LIN {X 0,Y 578.138,Z 351.984,A -85,B 0,C 180,E1 -8144.655,E2 -8144.655} C_VEL
LIN {X 0,Y 589.312,Z 368.246,A -85,B 0,C 180,E1 -8146.023,E2 -8146.023} C_VEL
LIN {X 0,Y 600.363,Z 385.488,A -85,B 0,C 180,E1 -8147.316,E2 -8147.316} C_VEL
LIN {X 0,Y 611.824,Z 404.452,A -85,B 0,C 180,E1 -8148.598,E2 -8148.598} C_VEL
LIN {X 0,Y 607.927,Z 580.681,A -85,B 0,C 180,E1 -8150.957,E2 -8150.957} C_VEL
LIN {X 0,Y 606.964,Z 588.376,A -85,B 0,C 180,E1 -8150.998,E2 -8150.998} C_VEL
LIN {X 0,Y 601.697,Z 608.927,A -85,B 0,C 180,E1 -8150.899,E2 -8150.899} C_VEL
LIN {X 0,Y 600.953,Z 615.53,A -85,B 0,C 180,E1 -8150.94,E2 -8150.94} C_VEL
LIN {X 0,Y 598.061,Z 740.001,A -85,B 0,C 180,E1 -8152.62,E2 -8152.62} C_VEL
LIN {X 0,Y 596.803,Z 765.646,A -85,B 0,C 180,E1 -8153.13,E2 -8153.13} C_VEL
LIN {X 0,Y 595.43,Z 786.189,A -85,B 0,C 180,E1 -8153.679,E2 -8153.679} C_VEL
LIN {X 0,Y 593.589,Z 809.668,A -85,B 0,C 180,E1 -8154.469,E2 -8154.469} C_VEL
LIN {X 0,Y 591.578,Z 830.485,A -85,B 0,C 180,E1 -8155.337,E2 -8155.337} C_VEL
LIN {X 0,Y 589.587,Z 849.41,A -85,B 0,C 180,E1 -8156.261,E2 -8156.261} C_VEL
LIN {X 0,Y 586.878,Z 872.633,A -85,B 0,C 180,E1 -8157.6,E2 -8157.6} C_VEL
LIN {X 0,Y 584.577,Z 891.053,A -85,B 0,C 180,E1 -8158.841,E2 -8158.841} C_VEL
LIN {X 0,Y 581.818,Z 912.391,A -85,B 0,C 180,E1 -8160.504,E2 -8160.504} C_VEL
LIN {X 0,Y 579.555,Z 929.188,A -85,B 0,C 180,E1 -8162.013,E2 -8162.013} C_VEL
LIN {X 0,Y 577.237,Z 946.768,A -85,B 0,C 180,E1 -8163.803,E2 -8163.803} C_VEL
LIN {X 0,Y 575.136,Z 962.606,A -85,B 0,C 180,E1 -8165.668,E2 -8165.668} C_VEL
LIN {X 0,Y 573.215,Z 978.266,A -85,B 0,C 180,E1 -8167.758,E2 -8167.758} C_VEL
LIN {X 0,Y 571.639,Z 991.661,A -85,B 0,C 180,E1 -8169.844,E2 -8169.844} C_VEL
LIN {X 0,Y 570.407,Z 1003.981,A -85,B 0,C 180,E1 -8172.03,E2 -8172.03} C_VEL
LIN {X 0,Y 569.421,Z 1014.821,A -85,B 0,C 180,E1 -8174.311,E2 -8174.311} C_VEL
LIN {X 0,Y 568.777,Z 1023.654,A -85,B 0,C 180,E1 -8176.479,E2 -8176.479} C_VEL
LIN {X 0,Y 568.305,Z 1031.896,A -85,B 0,C 180,E1 -8178.944,E2 -8178.944} C_VEL
LIN {X 0,Y 568.068,Z 1037.665,A -85,B 0,C 180,E1 -8181.089,E2 -8181.089} C_VEL
LIN {X 0,Y 567.957,Z 1042.942,A -85,B 0,C 180,E1 -8183.632,E2 -8183.632} C_VEL
LIN {X 0,Y 567.921,Z 1046.069,A -85,B 0,C 180,E1 -8185.861,E2 -8185.861} C_VEL
LIN {X 0,Y 567.907,Z 1047.939,A -85,B 0,C 180,E1 -8188.083,E2 -8188.083} C_VEL
LIN {X 0,Y 567.895,Z 1048.403,A -85,B 0,C 180,E1 -8190.504,E2 -8190.504} C_VEL
LIN {X 0,Y 567.903,Z 1047.524,A -85,B 0,C 180,E1 -8192.624,E2 -8192.624} C_VEL
LIN {X 0,Y 567.926,Z 1045.262,A -85,B 0,C 180,E1 -8194.949,E2 -8194.949} C_VEL
LIN {X 0,Y 567.983,Z 1041.193,A -85,B 0,C 180,E1 -8197.384,E2 -8197.384} C_VEL
LIN {X 0,Y 568.142,Z 1036.134,A -85,B 0,C 180,E1 -8199.625,E2 -8199.625} C_VEL
LIN {X 0,Y 568.484,Z 1028.635,A -85,B 0,C 180,E1 -8202.185,E2 -8202.185} C_VEL
LIN {X 0,Y 568.938,Z 1021.207,A -85,B 0,C 180,E1 -8204.244,E2 -8204.244} C_VEL
LIN {X 0,Y 569.749,Z 1011.047,A -85,B 0,C 180,E1 -8206.622,E2 -8206.622} C_VEL
LIN {X 0,Y 570.711,Z 1000.496,A -85,B 0,C 180,E1 -8208.7,E2 -8208.7} C_VEL
LIN {X 0,Y 572.024,Z 988.423,A -85,B 0,C 180,E1 -8210.784,E2 -8210.784} C_VEL
LIN {X 0,Y 573.664,Z 974.366,A -85,B 0,C 180,E1 -8212.873,E2 -8212.873} C_VEL
LIN {X 0,Y 575.487,Z 959.948,A -85,B 0,C 180,E1 -8214.754,E2 -8214.754} C_VEL
LIN {X 0,Y 577.795,Z 942.371,A -85,B 0,C 180,E1 -8216.753,E2 -8216.753} C_VEL
LIN {X 0,Y 579.967,Z 926.22,A -85,B 0,C 180,E1 -8218.358,E2 -8218.358} C_VEL
LIN {X 0,Y 582.671,Z 905.8,A -85,B 0,C 180,E1 -8220.13,E2 -8220.13} C_VEL
LIN {X 0,Y 584.966,Z 888.01,A -85,B 0,C 180,E1 -8221.466,E2 -8221.466} C_VEL
LIN {X 0,Y 587.578,Z 867.251,A -85,B 0,C 180,E1 -8222.827,E2 -8222.827} C_VEL
LIN {X 0,Y 589.85,Z 846.961,A -85,B 0,C 180,E1 -8223.956,E2 -8223.956} C_VEL
LIN {X 0,Y 591.882,Z 827.721,A -85,B 0,C 180,E1 -8224.879,E2 -8224.879} C_VEL
LIN {X 0,Y 594.088,Z 803.301,A -85,B 0,C 180,E1 -8225.853,E2 -8225.853} C_VEL
LIN {X 0,Y 595.735,Z 781.915,A -85,B 0,C 180,E1 -8226.539,E2 -8226.539} C_VEL
LIN {X 0,Y 597.341,Z 755.966,A -85,B 0,C 180,E1 -8227.177,E2 -8227.177} C_VEL
LIN {X 0,Y 598.277,Z 733.871,A -85,B 0,C 180,E1 -8227.564,E2 -8227.564} C_VEL
LIN {X 0,Y 603.923,Z 487.26,A -85,B 0,C 180,E1 -8230.874,E2 -8230.874} C_VEL
LIN {X 0,Y 605.687,Z 407.522,A -85,B 0,C 180,E1 -8231.966,E2 -8231.966} C_VEL
LIN {X 0,Y 591.197,Z 383.616,A -85,B 0,C 180,E1 -8233.642,E2 -8233.642} C_VEL
LIN {X 0,Y 577.413,Z 362.935,A -85,B 0,C 180,E1 -8235.327,E2 -8235.327} C_VEL
LIN {X 0,Y 571.826,Z 355.174,A -85,B 0,C 180,E1 -8236.037,E2 -8236.037} C_VEL
LIN {X 0,Y 569.839,Z 352.302,A -85,B 0,C 180,E1 -8236.297,E2 -8236.297} C_VEL
LIN {X 0,Y 569.32,Z 350.311,A -85,B 0,C 180,E1 -8236.561,E2 -8236.561} C_VEL
LIN {X 0,Y 569.374,Z 350.27,A -85,B 0,C 180,E1 -8239.81,E2 -8239.81} C_VEL
LIN {X 0,Y 569.32,Z 350.302,A -85,B 0,C 180,E1 -8242.878,E2 -8242.878} C_VEL
LIN {X 0,Y 569.348,Z 350.301,A -85,B 0,C 180,E1 -8246.171,E2 -8246.171} C_VEL
LIN {X 0,Y 569.335,Z 350.299,A -85,B 0,C 180,E1 -8249.265,E2 -8249.265} C_VEL
LIN {X 0,Y 569.322,Z 350.296,A -85,B 0,C 180,E1 -8252.603,E2 -8252.603} C_VEL
LIN {X 0,Y 569.371,Z 350.295,A -85,B 0,C 180,E1 -8255.736,E2 -8255.736} C_VEL
LIN {X 0,Y 569.317,Z 350.311,A -85,B 0,C 180,E1 -8258.897,E2 -8258.897} C_VEL
LIN {X 0,Y 569.379,Z 350.309,A -85,B 0,C 180,E1 -8262.102,E2 -8262.102} C_VEL
LIN {X 0,Y 569.316,Z 350.297,A -85,B 0,C 180,E1 -8265.246,E2 -8265.246} C_VEL
LIN {X 0,Y 569.348,Z 350.292,A -85,B 0,C 180,E1 -8268.511,E2 -8268.511} C_VEL
LIN {X 0,Y 569.334,Z 350.313,A -85,B 0,C 180,E1 -8271.618,E2 -8271.618} C_VEL
LIN {X 0,Y 569.322,Z 350.306,A -85,B 0,C 180,E1 -8274.962,E2 -8274.962} C_VEL
LIN {X 0,Y 569.367,Z 350.291,A -85,B 0,C 180,E1 -8278.088,E2 -8278.088} C_VEL
LIN {X 0,Y 569.319,Z 350.31,A -85,B 0,C 180,E1 -8281.208,E2 -8281.208} C_VEL
LIN {X 0,Y 569.376,Z 350.299,A -85,B 0,C 180,E1 -8284.432,E2 -8284.432} C_VEL
LIN {X 0,Y 569.315,Z 350.296,A -85,B 0,C 180,E1 -8287.569,E2 -8287.569} C_VEL
LIN {X 0,Y 569.354,Z 350.303,A -85,B 0,C 180,E1 -8290.831,E2 -8290.831} C_VEL
LIN {X 0,Y 569.327,Z 350.307,A -85,B 0,C 180,E1 -8293.923,E2 -8293.923} C_VEL
LIN {X 0,Y 569.326,Z 350.3,A -85,B 0,C 180,E1 -8297.266,E2 -8297.266} C_VEL
LIN {X 0,Y 569.356,Z 350.294,A -85,B 0,C 180,E1 -8300.348,E2 -8300.348} C_VEL
LIN {X 0,Y 569.319,Z 350.306,A -85,B 0,C 180,E1 -8303.54,E2 -8303.54} C_VEL
LIN {X 0,Y 569.38,Z 350.304,A -85,B 0,C 180,E1 -8306.716,E2 -8306.716} C_VEL
LIN {X 0,Y 569.316,Z 350.314,A -85,B 0,C 180,E1 -8309.818,E2 -8309.818} C_VEL
LIN {X 0,Y 569.377,Z 350.309,A -85,B 0,C 180,E1 -8312.984,E2 -8312.984} C_VEL
LIN {X 0,Y 569.321,Z 350.314,A -85,B 0,C 180,E1 -8316.165,E2 -8316.165} C_VEL
LIN {X 0,Y 569.336,Z 350.286,A -85,B 0,C 180,E1 -8319.477,E2 -8319.477} C_VEL
LIN {X 0,Y 569.374,Z 350.396,A -85,B 0,C 180,E1 -8321.295,E2 -8321.295} C_VEL
LIN {X 0,Y 570.486,Z 353.55,A -85,B 0,C 180,E1 -8321.761,E2 -8321.761} C_VEL
LIN {X 0,Y 574.758,Z 363.448,A -85,B 0,C 180,E1 -8323.27,E2 -8323.27} C_VEL
LIN {X 0,Y 579.045,Z 373.422,A -85,B 0,C 180,E1 -8324.688,E2 -8324.688} C_VEL
LIN {X 0,Y 591.062,Z 392.514,A -85,B 0,C 180,E1 -8326.162,E2 -8326.162} C_VEL
LIN {X 0,Y 603.404,Z 413.335,A -85,B 0,C 180,E1 -8327.599,E2 -8327.599} C_VEL
LIN {X 0,Y 605.024,Z 416.723,A -85,B 0,C 180,E1 -8327.791,E2 -8327.791} C_VEL
LIN {X 0,Y 605.75,Z 421.294,A -85,B 0,C 180,E1 -8327.924,E2 -8327.924} C_VEL
LIN {X 0,Y 599.74,Z 683.442,A -85,B 0,C 180,E1 -8331.446,E2 -8331.446} C_VEL
LIN {X 0,Y 597.787,Z 766.181,A -85,B 0,C 180,E1 -8332.567,E2 -8332.567} C_VEL
LIN {X 0,Y 596.415,Z 791.727,A -85,B 0,C 180,E1 -8333.073,E2 -8333.073} C_VEL
LIN {X 0,Y 594.909,Z 813.335,A -85,B 0,C 180,E1 -8333.649,E2 -8333.649} C_VEL
LIN {X 0,Y 592.891,Z 837.719,A -85,B 0,C 180,E1 -8334.48,E2 -8334.48} C_VEL
LIN {X 0,Y 590.939,Z 857.805,A -85,B 0,C 180,E1 -8335.319,E2 -8335.319} C_VEL
LIN {X 0,Y 588.667,Z 879.368,A -85,B 0,C 180,E1 -8336.376,E2 -8336.376} C_VEL
LIN {X 0,Y 586.06,Z 901.334,A -85,B 0,C 180,E1 -8337.665,E2 -8337.665} C_VEL
LIN {X 0,Y 583.558,Z 922.02,A -85,B 0,C 180,E1 -8339.067,E2 -8339.067} C_VEL
LIN {X 0,Y 581.019,Z 941.728,A -85,B 0,C 180,E1 -8340.629,E2 -8340.629} C_VEL
LIN {X 0,Y 578.772,Z 959.17,A -85,B 0,C 180,E1 -8342.196,E2 -8342.196} C_VEL
LIN {X 0,Y 576.449,Z 977.44,A -85,B 0,C 180,E1 -8344.08,E2 -8344.08} C_VEL
LIN {X 0,Y 574.58,Z 992.62,A -85,B 0,C 180,E1 -8345.861,E2 -8345.861} C_VEL
LIN {X 0,Y 572.692,Z 1008.993,A -85,B 0,C 180,E1 -8348.06,E2 -8348.06} C_VEL
LIN {X 0,Y 571.321,Z 1021.71,A -85,B 0,C 180,E1 -8350.023,E2 -8350.023} C_VEL
LIN {X 0,Y 570.111,Z 1034.752,A -85,B 0,C 180,E1 -8352.337,E2 -8352.337} C_VEL
LIN {X 0,Y 569.305,Z 1044.738,A -85,B 0,C 180,E1 -8354.412,E2 -8354.412} C_VEL
LIN {X 0,Y 568.673,Z 1054.559,A -85,B 0,C 180,E1 -8356.787,E2 -8356.787} C_VEL
LIN {X 0,Y 568.282,Z 1062.132,A -85,B 0,C 180,E1 -8359.053,E2 -8359.053} C_VEL
LIN {X 0,Y 568.057,Z 1067.991,A -85,B 0,C 180,E1 -8361.191,E2 -8361.191} C_VEL
LIN {X 0,Y 567.95,Z 1073.173,A -85,B 0,C 180,E1 -8363.733,E2 -8363.733} C_VEL
LIN {X 0,Y 567.913,Z 1076.121,A -85,B 0,C 180,E1 -8365.86,E2 -8365.86} C_VEL
LIN {X 0,Y 567.903,Z 1077.969,A -85,B 0,C 180,E1 -8368.083,E2 -8368.083} C_VEL
LIN {X 0,Y 567.895,Z 1078.393,A -85,B 0,C 180,E1 -8370.504,E2 -8370.504} C_VEL
LIN {X 0,Y 567.907,Z 1077.493,A -85,B 0,C 180,E1 -8372.624,E2 -8372.624} C_VEL
LIN {X 0,Y 567.93,Z 1075.211,A -85,B 0,C 180,E1 -8374.949,E2 -8374.949} C_VEL
LIN {X 0,Y 567.988,Z 1071.102,A -85,B 0,C 180,E1 -8377.383,E2 -8377.383} C_VEL
LIN {X 0,Y 568.109,Z 1066.7,A -85,B 0,C 180,E1 -8379.318,E2 -8379.318} C_VEL
LIN {X 0,Y 568.39,Z 1059.935,A -85,B 0,C 180,E1 -8381.672,E2 -8381.672} C_VEL
LIN {X 0,Y 568.853,Z 1051.422,A -85,B 0,C 180,E1 -8384.005,E2 -8384.005} C_VEL
LIN {X 0,Y 569.526,Z 1041.951,A -85,B 0,C 180,E1 -8386.209,E2 -8386.209} C_VEL
LIN {X 0,Y 570.517,Z 1030.092,A -85,B 0,C 180,E1 -8388.529,E2 -8388.529} C_VEL
LIN {X 0,Y 571.653,Z 1018.636,A -85,B 0,C 180,E1 -8390.476,E2 -8390.476} C_VEL
LIN {X 0,Y 573.354,Z 1003.039,A -85,B 0,C 180,E1 -8392.777,E2 -8392.777} C_VEL
LIN {X 0,Y 575.002,Z 989.119,A -85,B 0,C 180,E1 -8394.568,E2 -8394.568} C_VEL
LIN {X 0,Y 577.243,Z 971.153,A -85,B 0,C 180,E1 -8396.601,E2 -8396.601} C_VEL
LIN {X 0,Y 579.35,Z 954.693,A -85,B 0,C 180,E1 -8398.222,E2 -8398.222} C_VEL
LIN {X 0,Y 581.834,Z 935.535,A -85,B 0,C 180,E1 -8399.892,E2 -8399.892} C_VEL
LIN {X 0,Y 584.258,Z 916.056,A -85,B 0,C 180,E1 -8401.352,E2 -8401.352} C_VEL
LIN {X 0,Y 586.8,Z 895.61,A -85,B 0,C 180,E1 -8402.694,E2 -8402.694} C_VEL
LIN {X 0,Y 589.267,Z 873.458,A -85,B 0,C 180,E1 -8403.926,E2 -8403.926} C_VEL
LIN {X 0,Y 591.337,Z 853.89,A -85,B 0,C 180,E1 -8404.856,E2 -8404.856} C_VEL
LIN {X 0,Y 593.584,Z 829.334,A -85,B 0,C 180,E1 -8405.828,E2 -8405.828} C_VEL
LIN {X 0,Y 595.294,Z 807.859,A -85,B 0,C 180,E1 -8406.51,E2 -8406.51} C_VEL
LIN {X 0,Y 597.016,Z 781.97,A -85,B 0,C 180,E1 -8407.14,E2 -8407.14} C_VEL
LIN {X 0,Y 597.994,Z 759.969,A -85,B 0,C 180,E1 -8407.525,E2 -8407.525} C_VEL
LIN {X 0,Y 603.364,Z 520.75,A -85,B 0,C 180,E1 -8410.732,E2 -8410.732} C_VEL
LIN {X 0,Y 605.608,Z 419.549,A -85,B 0,C 180,E1 -8412.111,E2 -8412.111} C_VEL
LIN {X 0,Y 604.432,Z 415.199,A -85,B 0,C 180,E1 -8412.279,E2 -8412.279} C_VEL
LIN {X 0,Y 592.065,Z 394.2,A -85,B 0,C 180,E1 -8413.712,E2 -8413.712} C_VEL
LIN {X 0,Y 581.887,Z 377.919,A -85,B 0,C 180,E1 -8414.948,E2 -8414.948} C_VEL
LIN {X 0,Y 578.649,Z 372.548,A -85,B 0,C 180,E1 -8415.392,E2 -8415.392} C_VEL
LIN {X 0,Y 572.311,Z 357.615,A -85,B 0,C 180,E1 -8417.593,E2 -8417.593} C_VEL
LIN {X 0,Y 569.389,Z 350.526,A -85,B 0,C 180,E1 -8418.678,E2 -8418.678} C_VEL
LIN {X 0,Y 569.319,Z 350.311,A -85,B 0,C 180,E1 -8421.889,E2 -8421.889} C_VEL
LIN {X 0,Y 569.372,Z 350.251,A -85,B 0,C 180,E1 -8425.096,E2 -8425.096} C_VEL
LIN {X 0,Y 569.315,Z 350.302,A -85,B 0,C 180,E1 -8428.217,E2 -8428.217} C_VEL
LIN {X 0,Y 569.376,Z 350.295,A -85,B 0,C 180,E1 -8431.409,E2 -8431.409} C_VEL
LIN {X 0,Y 569.332,Z 350.309,A -85,B 0,C 180,E1 -8434.626,E2 -8434.626} C_VEL
LIN {X 0,Y 569.326,Z 350.312,A -85,B 0,C 180,E1 -8438.032,E2 -8438.032} C_VEL
LIN {X 0,Y 569.37,Z 350.301,A -85,B 0,C 180,E1 -8441.183,E2 -8441.183} C_VEL
LIN {X 0,Y 569.317,Z 350.3,A -85,B 0,C 180,E1 -8444.412,E2 -8444.412} C_VEL
LIN {X 0,Y 569.38,Z 350.294,A -85,B 0,C 180,E1 -8447.526,E2 -8447.526} C_VEL
LIN {X 0,Y 569.321,Z 350.31,A -85,B 0,C 180,E1 -8450.701,E2 -8450.701} C_VEL
LIN {X 0,Y 569.355,Z 350.3,A -85,B 0,C 180,E1 -8453.951,E2 -8453.951} C_VEL
LIN {X 0,Y 569.335,Z 350.294,A -85,B 0,C 180,E1 -8457.081,E2 -8457.081} C_VEL
LIN {X 0,Y 569.328,Z 350.307,A -85,B 0,C 180,E1 -8460.403,E2 -8460.403} C_VEL
LIN {X 0,Y 569.368,Z 350.299,A -85,B 0,C 180,E1 -8463.524,E2 -8463.524} C_VEL
LIN {X 0,Y 569.319,Z 350.292,A -85,B 0,C 180,E1 -8466.758,E2 -8466.758} C_VEL
LIN {X 0,Y 569.382,Z 350.303,A -85,B 0,C 180,E1 -8469.91,E2 -8469.91} C_VEL
LIN {X 0,Y 569.325,Z 350.309,A -85,B 0,C 180,E1 -8473.095,E2 -8473.095} C_VEL
LIN {X 0,Y 569.359,Z 350.294,A -85,B 0,C 180,E1 -8476.319,E2 -8476.319} C_VEL
LIN {X 0,Y 569.337,Z 350.302,A -85,B 0,C 180,E1 -8479.422,E2 -8479.422} C_VEL
LIN {X 0,Y 569.332,Z 350.307,A -85,B 0,C 180,E1 -8482.775,E2 -8482.775} C_VEL
LIN {X 0,Y 569.374,Z 350.307,A -85,B 0,C 180,E1 -8485.956,E2 -8485.956} C_VEL
LIN {X 0,Y 569.325,Z 350.312,A -85,B 0,C 180,E1 -8489.207,E2 -8489.207} C_VEL
LIN {X 0,Y 569.38,Z 350.299,A -85,B 0,C 180,E1 -8492.386,E2 -8492.386} C_VEL
LIN {X 0,Y 569.332,Z 350.308,A -85,B 0,C 180,E1 -8495.596,E2 -8495.596} C_VEL
LIN {X 0,Y 569.341,Z 350.314,A -85,B 0,C 180,E1 -8498.957,E2 -8498.957} C_VEL
LIN {X 0,Y 569.358,Z 350.309,A -85,B 0,C 180,E1 -8502.024,E2 -8502.024} C_VEL
LIN {X 0,Y 569.352,Z 350.49,A -85,B 0,C 180,E1 -8503.584,E2 -8503.584} C_VEL
LIN {X 0,Y 569.857,Z 352.317,A -85,B 0,C 180,E1 -8503.805,E2 -8503.805} C_VEL
LIN {X 0,Y 571.834,Z 355.169,A -85,B 0,C 180,E1 -8504.063,E2 -8504.063} C_VEL
LIN {X 0,Y 582.055,Z 369.753,A -85,B 0,C 180,E1 -8505.35,E2 -8505.35} C_VEL
LIN {X 0,Y 594.983,Z 389.805,A -85,B 0,C 180,E1 -8506.903,E2 -8506.903} C_VEL
LIN {X 0,Y 605.783,Z 407.826,A -85,B 0,C 180,E1 -8508.141,E2 -8508.141} C_VEL
LIN {X 0,Y 600.953,Z 615.53,A -85,B 0,C 180,E1 -8510.94,E2 -8510.94} C_VEL
LIN {X 0,Y 599.989,Z 623.225,A -85,B 0,C 180,E1 -8510.982,E2 -8510.982} C_VEL
LIN {X 0,Y 594.69,Z 643.768,A -85,B 0,C 180,E1 -8510.878,E2 -8510.878} C_VEL
LIN {X 0,Y 593.943,Z 650.371,A -85,B 0,C 180,E1 -8510.92,E2 -8510.92} C_VEL
LIN {X 0,Y 591.701,Z 740.883,A -85,B 0,C 180,E1 -8512.159,E2 -8512.159} C_VEL
LIN {X 0,Y 590.392,Z 766.136,A -85,B 0,C 180,E1 -8512.669,E2 -8512.669} C_VEL
LIN {X 0,Y 588.954,Z 786.751,A -85,B 0,C 180,E1 -8513.226,E2 -8513.226} C_VEL
LIN {X 0,Y 587.053,Z 809.894,A -85,B 0,C 180,E1 -8514.012,E2 -8514.012} C_VEL
LIN {X 0,Y 584.956,Z 830.709,A -85,B 0,C 180,E1 -8514.887,E2 -8514.887} C_VEL
LIN {X 0,Y 582.871,Z 849.635,A -85,B 0,C 180,E1 -8515.819,E2 -8515.819} C_VEL
LIN {X 0,Y 580.033,Z 872.857,A -85,B 0,C 180,E1 -8517.17,E2 -8517.17} C_VEL
LIN {X 0,Y 577.624,Z 891.204,A -85,B 0,C 180,E1 -8518.418,E2 -8518.418} C_VEL
LIN {X 0,Y 574.802,Z 912.012,A -85,B 0,C 180,E1 -8520.05,E2 -8520.05} C_VEL
LIN {X 0,Y 572.415,Z 928.862,A -85,B 0,C 180,E1 -8521.576,E2 -8521.576} C_VEL
LIN {X 0,Y 569.967,Z 946.379,A -85,B 0,C 180,E1 -8523.368,E2 -8523.368} C_VEL
LIN {X 0,Y 567.657,Z 962.831,A -85,B 0,C 180,E1 -8525.326,E2 -8525.326} C_VEL
LIN {X 0,Y 565.703,Z 977.766,A -85,B 0,C 180,E1 -8527.337,E2 -8527.337} C_VEL
LIN {X 0,Y 564.021,Z 991.257,A -85,B 0,C 180,E1 -8529.451,E2 -8529.451} C_VEL
LIN {X 0,Y 562.712,Z 1003.072,A -85,B 0,C 180,E1 -8531.561,E2 -8531.561} C_VEL
LIN {X 0,Y 561.593,Z 1014.59,A -85,B 0,C 180,E1 -8533.98,E2 -8533.98} C_VEL
LIN {X 0,Y 560.919,Z 1023.076,A -85,B 0,C 180,E1 -8536.075,E2 -8536.075} C_VEL
LIN {X 0,Y 560.365,Z 1031.816,A -85,B 0,C 180,E1 -8538.681,E2 -8538.681} C_VEL
LIN {X 0,Y 560.107,Z 1037.632,A -85,B 0,C 180,E1 -8540.858,E2 -8540.858} C_VEL
LIN {X 0,Y 559.977,Z 1042.622,A -85,B 0,C 180,E1 -8543.232,E2 -8543.232} C_VEL
LIN {X 0,Y 559.925,Z 1046.063,A -85,B 0,C 180,E1 -8545.699,E2 -8545.699} C_VEL
LIN {X 0,Y 559.911,Z 1047.879,A -85,B 0,C 180,E1 -8547.851,E2 -8547.851} C_VEL
LIN {X 0,Y 559.896,Z 1048.491,A -85,B 0,C 180,E1 -8550.409,E2 -8550.409} C_VEL
LIN {X 0,Y 559.905,Z 1047.67,A -85,B 0,C 180,E1 -8552.559,E2 -8552.559} C_VEL
LIN {X 0,Y 559.926,Z 1045.716,A -85,B 0,C 180,E1 -8554.712,E2 -8554.712} C_VEL
LIN {X 0,Y 559.998,Z 1041.786,A -85,B 0,C 180,E1 -8557.283,E2 -8557.283} C_VEL
LIN {X 0,Y 560.142,Z 1037.098,A -85,B 0,C 180,E1 -8559.452,E2 -8559.452} C_VEL
LIN {X 0,Y 560.472,Z 1030.242,A -85,B 0,C 180,E1 -8561.943,E2 -8561.943} C_VEL
LIN {X 0,Y 560.979,Z 1022.221,A -85,B 0,C 180,E1 -8564.239,E2 -8564.239} C_VEL
LIN {X 0,Y 561.731,Z 1013.16,A -85,B 0,C 180,E1 -8566.441,E2 -8566.441} C_VEL
LIN {X 0,Y 562.829,Z 1001.843,A -85,B 0,C 180,E1 -8568.757,E2 -8568.757} C_VEL
LIN {X 0,Y 564.111,Z 990.519,A -85,B 0,C 180,E1 -8570.763,E2 -8570.763} C_VEL
LIN {X 0,Y 566.001,Z 975.343,A -85,B 0,C 180,E1 -8573.09,E2 -8573.09} C_VEL
LIN {X 0,Y 567.91,Z 960.999,A -85,B 0,C 180,E1 -8574.996,E2 -8574.996} C_VEL
LIN {X 0,Y 570.46,Z 942.701,A -85,B 0,C 180,E1 -8577.111,E2 -8577.111} C_VEL
LIN {X 0,Y 572.685,Z 926.983,A -85,B 0,C 180,E1 -8578.695,E2 -8578.695} C_VEL
LIN {X 0,Y 575.36,Z 908.011,A -85,B 0,C 180,E1 -8580.379,E2 -8580.379} C_VEL
LIN {X 0,Y 577.956,Z 888.775,A -85,B 0,C 180,E1 -8581.848,E2 -8581.848} C_VEL
LIN {X 0,Y 580.71,Z 867.993,A -85,B 0,C 180,E1 -8583.23,E2 -8583.23} C_VEL
LIN {X 0,Y 583.147,Z 847.168,A -85,B 0,C 180,E1 -8584.401,E2 -8584.401} C_VEL
LIN {X 0,Y 585.274,Z 827.927,A -85,B 0,C 180,E1 -8585.331,E2 -8585.331} C_VEL
LIN {X 0,Y 587.577,Z 803.504,A -85,B 0,C 180,E1 -8586.313,E2 -8586.313} C_VEL
LIN {X 0,Y 589.299,Z 782.115,A -85,B 0,C 180,E1 -8587.004,E2 -8587.004} C_VEL
LIN {X 0,Y 590.996,Z 755.836,A -85,B 0,C 180,E1 -8587.653,E2 -8587.653} C_VEL
LIN {X 0,Y 591.96,Z 733.844,A -85,B 0,C 180,E1 -8588.04,E2 -8588.04} C_VEL
LIN {X 0,Y 597.916,Z 486.426,A -85,B 0,C 180,E1 -8591.39,E2 -8591.39} C_VEL
LIN {X 0,Y 599.668,Z 410.831,A -85,B 0,C 180,E1 -8592.435,E2 -8592.435} C_VEL
LIN {X 0,Y 585.558,Z 387.591,A -85,B 0,C 180,E1 -8594.107,E2 -8594.107} C_VEL
LIN {X 0,Y 572.751,Z 368.31,A -85,B 0,C 180,E1 -8595.708,E2 -8595.708} C_VEL
LIN {X 0,Y 567.821,Z 361.432,A -85,B 0,C 180,E1 -8596.347,E2 -8596.347} C_VEL
LIN {X 0,Y 565.177,Z 357.429,A -85,B 0,C 180,E1 -8596.703,E2 -8596.703} C_VEL
LIN {X 0,Y 562.249,Z 353.997,A -85,B 0,C 180,E1 -8597.086,E2 -8597.086} C_VEL
LIN {X 0,Y 561.547,Z 352.059,A -85,B 0,C 180,E1 -8597.211,E2 -8597.211} C_VEL
LIN {X 0,Y 561.423,Z 351.263,A -85,B 0,C 180,E1 -8597.354,E2 -8597.354} C_VEL
LIN {X 0,Y 561.38,Z 351.286,A -85,B 0,C 180,E1 -8600.516,E2 -8600.516} C_VEL
LIN {X 0,Y 561.44,Z 351.29,A -85,B 0,C 180,E1 -8603.626,E2 -8603.626} C_VEL
LIN {X 0,Y 561.38,Z 351.299,A -85,B 0,C 180,E1 -8606.852,E2 -8606.852} C_VEL
LIN {X 0,Y 561.42,Z 351.297,A -85,B 0,C 180,E1 -8610.152,E2 -8610.152} C_VEL
LIN {X 0,Y 561.387,Z 351.288,A -85,B 0,C 180,E1 -8613.216,E2 -8613.216} C_VEL
LIN {X 0,Y 561.388,Z 351.286,A -85,B 0,C 180,E1 -8616.597,E2 -8616.597} C_VEL
LIN {X 0,Y 561.407,Z 351.288,A -85,B 0,C 180,E1 -8619.569,E2 -8619.569} C_VEL
LIN {X 0,Y 561.383,Z 351.299,A -85,B 0,C 180,E1 -8622.802,E2 -8622.802} C_VEL
LIN {X 0,Y 561.446,Z 351.288,A -85,B 0,C 180,E1 -8625.983,E2 -8625.983} C_VEL
LIN {X 0,Y 561.377,Z 351.281,A -85,B 0,C 180,E1 -8629.221,E2 -8629.221} C_VEL
LIN {X 0,Y 561.415,Z 351.288,A -85,B 0,C 180,E1 -8632.53,E2 -8632.53} C_VEL
LIN {X 0,Y 561.39,Z 351.298,A -85,B 0,C 180,E1 -8635.608,E2 -8635.608} C_VEL
LIN {X 0,Y 561.385,Z 351.285,A -85,B 0,C 180,E1 -8638.979,E2 -8638.979} C_VEL
LIN {X 0,Y 561.417,Z 351.287,A -85,B 0,C 180,E1 -8642.041,E2 -8642.041} C_VEL
LIN {X 0,Y 561.379,Z 351.3,A -85,B 0,C 180,E1 -8645.344,E2 -8645.344} C_VEL
LIN {X 0,Y 561.443,Z 351.281,A -85,B 0,C 180,E1 -8648.5,E2 -8648.5} C_VEL
LIN {X 0,Y 561.38,Z 351.289,A -85,B 0,C 180,E1 -8651.715,E2 -8651.715} C_VEL
LIN {X 0,Y 561.4,Z 351.294,A -85,B 0,C 180,E1 -8655.072,E2 -8655.072} C_VEL
LIN {X 0,Y 561.4,Z 351.294,A -85,B 0,C 180,E1 -8658.161,E2 -8658.161} C_VEL
LIN {X 0,Y 561.383,Z 351.29,A -85,B 0,C 180,E1 -8661.416,E2 -8661.416} C_VEL
LIN {X 0,Y 561.427,Z 351.281,A -85,B 0,C 180,E1 -8664.517,E2 -8664.517} C_VEL
LIN {X 0,Y 561.378,Z 351.29,A -85,B 0,C 180,E1 -8667.721,E2 -8667.721} C_VEL
LIN {X 0,Y 561.447,Z 351.284,A -85,B 0,C 180,E1 -8670.862,E2 -8670.862} C_VEL
LIN {X 0,Y 561.381,Z 351.293,A -85,B 0,C 180,E1 -8674.083,E2 -8674.083} C_VEL
LIN {X 0,Y 561.403,Z 351.291,A -85,B 0,C 180,E1 -8677.406,E2 -8677.406} C_VEL
LIN {X 0,Y 561.388,Z 351.255,A -85,B 0,C 180,E1 -8680.415,E2 -8680.415} C_VEL
LIN {X 0,Y 561.459,Z 351.65,A -85,B 0,C 180,E1 -8680.543,E2 -8680.543} C_VEL
LIN {X 0,Y 568.29,Z 367.681,A -85,B 0,C 180,E1 -8683.053,E2 -8683.053} C_VEL
LIN {X 0,Y 570.669,Z 373.151,A -85,B 0,C 180,E1 -8683.831,E2 -8683.831} C_VEL
LIN {X 0,Y 585.664,Z 396.661,A -85,B 0,C 180,E1 -8685.725,E2 -8685.725} C_VEL
LIN {X 0,Y 599.017,Z 419.466,A -85,B 0,C 180,E1 -8687.314,E2 -8687.314} C_VEL
LIN {X 0,Y 599.771,Z 422.469,A -85,B 0,C 180,E1 -8687.428,E2 -8687.428} C_VEL
LIN {X 0,Y 593.459,Z 684.126,A -85,B 0,C 180,E1 -8690.974,E2 -8690.974} C_VEL
LIN {X 0,Y 591.429,Z 765.982,A -85,B 0,C 180,E1 -8692.094,E2 -8692.094} C_VEL
LIN {X 0,Y 589.985,Z 791.636,A -85,B 0,C 180,E1 -8692.606,E2 -8692.606} C_VEL
LIN {X 0,Y 588.396,Z 813.431,A -85,B 0,C 180,E1 -8693.192,E2 -8693.192} C_VEL
LIN {X 0,Y 586.304,Z 837.508,A -85,B 0,C 180,E1 -8694.019,E2 -8694.019} C_VEL
LIN {X 0,Y 584.314,Z 857.114,A -85,B 0,C 180,E1 -8694.843,E2 -8694.843} C_VEL
LIN {X 0,Y 581.985,Z 878.145,A -85,B 0,C 180,E1 -8695.879,E2 -8695.879} C_VEL
LIN {X 0,Y 579.255,Z 900.301,A -85,B 0,C 180,E1 -8697.179,E2 -8697.179} C_VEL
LIN {X 0,Y 576.768,Z 919.582,A -85,B 0,C 180,E1 -8698.488,E2 -8698.488} C_VEL
LIN {X 0,Y 574,Z 940.283,A -85,B 0,C 180,E1 -8700.119,E2 -8700.119} C_VEL
LIN {X 0,Y 571.693,Z 957.27,A -85,B 0,C 180,E1 -8701.65,E2 -8701.65} C_VEL
LIN {X 0,Y 569.073,Z 976.648,A -85,B 0,C 180,E1 -8703.65,E2 -8703.65} C_VEL
LIN {X 0,Y 567.125,Z 991.544,A -85,B 0,C 180,E1 -8705.412,E2 -8705.412} C_VEL
LIN {X 0,Y 565.179,Z 1007.354,A -85,B 0,C 180,E1 -8707.534,E2 -8707.534} C_VEL
LIN {X 0,Y 563.688,Z 1020.339,A -85,B 0,C 180,E1 -8709.547,E2 -8709.547} C_VEL
LIN {X 0,Y 562.421,Z 1032.952,A -85,B 0,C 180,E1 -8711.766,E2 -8711.766} C_VEL
LIN {X 0,Y 561.428,Z 1044.126,A -85,B 0,C 180,E1 -8714.098,E2 -8714.098} C_VEL
LIN {X 0,Y 560.777,Z 1053.404,A -85,B 0,C 180,E1 -8716.352,E2 -8716.352} C_VEL
LIN {X 0,Y 560.317,Z 1061.584,A -85,B 0,C 180,E1 -8718.784,E2 -8718.784} C_VEL
LIN {X 0,Y 560.084,Z 1067.259,A -85,B 0,C 180,E1 -8720.858,E2 -8720.858} C_VEL
LIN {X 0,Y 559.957,Z 1072.383,A -85,B 0,C 180,E1 -8723.232,E2 -8723.232} C_VEL
LIN {X 0,Y 559.916,Z 1075.802,A -85,B 0,C 180,E1 -8725.596,E2 -8725.596} C_VEL
LIN {X 0,Y 559.909,Z 1077.638,A -85,B 0,C 180,E1 -8727.646,E2 -8727.646} C_VEL
LIN {X 0,Y 559.907,Z 1078.437,A -85,B 0,C 180,E1 -8730.102,E2 -8730.102} C_VEL
LIN {X 0,Y 559.908,Z 1077.568,A -85,B 0,C 180,E1 -8732.456,E2 -8732.456} C_VEL
LIN {X 0,Y 559.921,Z 1075.57,A -85,B 0,C 180,E1 -8734.609,E2 -8734.609} C_VEL
LIN {X 0,Y 559.992,Z 1071.559,A -85,B 0,C 180,E1 -8737.18,E2 -8737.18} C_VEL
LIN {X 0,Y 560.113,Z 1066.743,A -85,B 0,C 180,E1 -8739.349,E2 -8739.349} C_VEL
LIN {X 0,Y 560.404,Z 1060.043,A -85,B 0,C 180,E1 -8741.736,E2 -8741.736} C_VEL
LIN {X 0,Y 560.897,Z 1051.486,A -85,B 0,C 180,E1 -8744.136,E2 -8744.136} C_VEL
LIN {X 0,Y 561.59,Z 1042.249,A -85,B 0,C 180,E1 -8746.327,E2 -8746.327} C_VEL
LIN {X 0,Y 562.677,Z 1030.057,A -85,B 0,C 180,E1 -8748.762,E2 -8748.762} C_VEL
LIN {X 0,Y 563.903,Z 1018.415,A -85,B 0,C 180,E1 -8750.771,E2 -8750.771} C_VEL
LIN {X 0,Y 565.719,Z 1002.818,A -85,B 0,C 180,E1 -8753.102,E2 -8753.102} C_VEL
LIN {X 0,Y 567.452,Z 988.983,A -85,B 0,C 180,E1 -8754.906,E2 -8754.906} C_VEL
LIN {X 0,Y 569.812,Z 971.192,A -85,B 0,C 180,E1 -8756.947,E2 -8756.947} C_VEL
LIN {X 0,Y 572.064,Z 954.471,A -85,B 0,C 180,E1 -8758.614,E2 -8758.614} C_VEL
LIN {X 0,Y 574.683,Z 935.312,A -85,B 0,C 180,E1 -8760.303,E2 -8760.303} C_VEL
LIN {X 0,Y 577.247,Z 915.868,A -85,B 0,C 180,E1 -8761.775,E2 -8761.775} C_VEL
LIN {X 0,Y 579.916,Z 895.388,A -85,B 0,C 180,E1 -8763.132,E2 -8763.132} C_VEL
LIN {X 0,Y 582.412,Z 874.076,A -85,B 0,C 180,E1 -8764.331,E2 -8764.331} C_VEL
LIN {X 0,Y 584.554,Z 854.804,A -85,B 0,C 180,E1 -8765.261,E2 -8765.261} C_VEL
LIN {X 0,Y 586.912,Z 830.596,A -85,B 0,C 180,E1 -8766.24,E2 -8766.24} C_VEL
LIN {X 0,Y 588.742,Z 808.674,A -85,B 0,C 180,E1 -8766.947,E2 -8766.947} C_VEL
LIN {X 0,Y 590.508,Z 783.929,A -85,B 0,C 180,E1 -8767.569,E2 -8767.569} C_VEL
LIN {X 0,Y 591.608,Z 760.704,A -85,B 0,C 180,E1 -8767.984,E2 -8767.984} C_VEL
LIN {X 0,Y 597.197,Z 524.469,A -85,B 0,C 180,E1 -8771.181,E2 -8771.181} C_VEL
LIN {X 0,Y 599.615,Z 421.343,A -85,B 0,C 180,E1 -8772.599,E2 -8772.599} C_VEL
LIN {X 0,Y 598.673,Z 418.87,A -85,B 0,C 180,E1 -8772.72,E2 -8772.72} C_VEL
LIN {X 0,Y 585.08,Z 395.729,A -85,B 0,C 180,E1 -8774.339,E2 -8774.339} C_VEL
LIN {X 0,Y 570.324,Z 372.582,A -85,B 0,C 180,E1 -8776.209,E2 -8776.209} C_VEL
LIN {X 0,Y 564.668,Z 359.074,A -85,B 0,C 180,E1 -8778.256,E2 -8778.256} C_VEL
LIN {X 0,Y 561.444,Z 351.567,A -85,B 0,C 180,E1 -8779.455,E2 -8779.455} C_VEL
LIN {X 0,Y 561.381,Z 351.293,A -85,B 0,C 180,E1 -8779.851,E2 -8779.851} C_VEL
LIN {X 0,Y 561.435,Z 351.252,A -85,B 0,C 180,E1 -8782.989,E2 -8782.989} C_VEL
LIN {X 0,Y 561.377,Z 351.277,A -85,B 0,C 180,E1 -8786.24,E2 -8786.24} C_VEL
LIN {X 0,Y 561.415,Z 351.284,A -85,B 0,C 180,E1 -8789.543,E2 -8789.543} C_VEL
LIN {X 0,Y 561.387,Z 351.282,A -85,B 0,C 180,E1 -8792.528,E2 -8792.528} C_VEL
LIN {X 0,Y 561.39,Z 351.285,A -85,B 0,C 180,E1 -8795.929,E2 -8795.929} C_VEL
LIN {X 0,Y 561.412,Z 351.292,A -85,B 0,C 180,E1 -8798.948,E2 -8798.948} C_VEL
LIN {X 0,Y 561.382,Z 351.299,A -85,B 0,C 180,E1 -8802.267,E2 -8802.267} C_VEL
LIN {X 0,Y 561.45,Z 351.289,A -85,B 0,C 180,E1 -8805.457,E2 -8805.457} C_VEL
LIN {X 0,Y 561.383,Z 351.285,A -85,B 0,C 180,E1 -8808.701,E2 -8808.701} C_VEL
LIN {X 0,Y 561.404,Z 351.281,A -85,B 0,C 180,E1 -8812.014,E2 -8812.014} C_VEL
LIN {X 0,Y 561.401,Z 351.298,A -85,B 0,C 180,E1 -8815.096,E2 -8815.096} C_VEL
LIN {X 0,Y 561.386,Z 351.294,A -85,B 0,C 180,E1 -8818.469,E2 -8818.469} C_VEL
LIN {X 0,Y 561.44,Z 351.279,A -85,B 0,C 180,E1 -8821.633,E2 -8821.633} C_VEL
LIN {X 0,Y 561.383,Z 351.299,A -85,B 0,C 180,E1 -8824.904,E2 -8824.904} C_VEL
LIN {X 0,Y 561.419,Z 351.291,A -85,B 0,C 180,E1 -8828.191,E2 -8828.191} C_VEL
LIN {X 0,Y 561.395,Z 351.28,A -85,B 0,C 180,E1 -8831.298,E2 -8831.298} C_VEL
LIN {X 0,Y 561.39,Z 351.292,A -85,B 0,C 180,E1 -8834.65,E2 -8834.65} C_VEL
LIN {X 0,Y 561.438,Z 351.294,A -85,B 0,C 180,E1 -8837.838,E2 -8837.838} C_VEL
LIN {X 0,Y 561.385,Z 351.296,A -85,B 0,C 180,E1 -8841.087,E2 -8841.087} C_VEL
LIN {X 0,Y 561.435,Z 351.281,A -85,B 0,C 180,E1 -8844.293,E2 -8844.293} C_VEL
LIN {X 0,Y 561.394,Z 351.287,A -85,B 0,C 180,E1 -8847.504,E2 -8847.504} C_VEL
LIN {X 0,Y 561.396,Z 351.286,A -85,B 0,C 180,E1 -8850.861,E2 -8850.861} C_VEL
LIN {X 0,Y 561.43,Z 351.288,A -85,B 0,C 180,E1 -8854.002,E2 -8854.002} C_VEL
LIN {X 0,Y 561.386,Z 351.288,A -85,B 0,C 180,E1 -8857.271,E2 -8857.271} C_VEL
LIN {X 0,Y 561.449,Z 351.284,A -85,B 0,C 180,E1 -8860.496,E2 -8860.496} C_VEL
LIN {X 0,Y 561.432,Z 351.385,A -85,B 0,C 180,E1 -8862.798,E2 -8862.798} C_VEL
LIN {X 0,Y 561.771,Z 352.874,A -85,B 0,C 180,E1 -8862.942,E2 -8862.942} C_VEL
LIN {X 0,Y 563.546,Z 355.831,A -85,B 0,C 180,E1 -8863.191,E2 -8863.191} C_VEL
LIN {X 0,Y 565.265,Z 357.608,A -85,B 0,C 180,E1 -8863.41,E2 -8863.41} C_VEL
LIN {X 0,Y 568,Z 361.604,A -85,B 0,C 180,E1 -8863.775,E2 -8863.775} C_VEL
LIN {X 0,Y 580.06,Z 379.111,A -85,B 0,C 180,E1 -8865.314,E2 -8865.314} C_VEL
LIN {X 0,Y 591.377,Z 397.055,A -85,B 0,C 180,E1 -8866.692,E2 -8866.692} C_VEL
LIN {X 0,Y 599.764,Z 411.252,A -85,B 0,C 180,E1 -8867.674,E2 -8867.674} C_VEL
LIN {X 0,Y 593.943,Z 650.371,A -85,B 0,C 180,E1 -8870.92,E2 -8870.92} C_VEL
LIN {X 0,Y 592.979,Z 658.066,A -85,B 0,C 180,E1 -8870.962,E2 -8870.962} C_VEL
LIN {X 0,Y 587.661,Z 678.606,A -85,B 0,C 180,E1 -8870.856,E2 -8870.856} C_VEL
LIN {X 0,Y 586.911,Z 685.209,A -85,B 0,C 180,E1 -8870.898,E2 -8870.898} C_VEL
LIN {X 0,Y 585.342,Z 743.046,A -85,B 0,C 180,E1 -8871.709,E2 -8871.709} C_VEL
LIN {X 0,Y 583.986,Z 767.146,A -85,B 0,C 180,E1 -8872.212,E2 -8872.212} C_VEL
LIN {X 0,Y 582.473,Z 787.884,A -85,B 0,C 180,E1 -8872.781,E2 -8872.781} C_VEL
LIN {X 0,Y 580.42,Z 811.398,A -85,B 0,C 180,E1 -8873.596,E2 -8873.596} C_VEL
LIN {X 0,Y 578.245,Z 832.059,A -85,B 0,C 180,E1 -8874.479,E2 -8874.479} C_VEL
LIN {X 0,Y 575.85,Z 852.856,A -85,B 0,C 180,E1 -8875.524,E2 -8875.524} C_VEL
LIN {X 0,Y 572.995,Z 874.718,A -85,B 0,C 180,E1 -8876.836,E2 -8876.836} C_VEL
LIN {X 0,Y 570.331,Z 894.157,A -85,B 0,C 180,E1 -8878.188,E2 -8878.188} C_VEL
LIN {X 0,Y 567.454,Z 914.045,A -85,B 0,C 180,E1 -8879.797,E2 -8879.797} C_VEL
LIN {X 0,Y 564.979,Z 930.736,A -85,B 0,C 180,E1 -8881.34,E2 -8881.34} C_VEL
LIN {X 0,Y 562.137,Z 949.831,A -85,B 0,C 180,E1 -8883.369,E2 -8883.369} C_VEL
LIN {X 0,Y 559.962,Z 964.727,A -85,B 0,C 180,E1 -8885.189,E2 -8885.189} C_VEL
LIN {X 0,Y 557.73,Z 980.79,A -85,B 0,C 180,E1 -8887.44,E2 -8887.44} C_VEL
LIN {X 0,Y 556.178,Z 992.734,A -85,B 0,C 180,E1 -8889.368,E2 -8889.368} C_VEL
LIN {X 0,Y 554.714,Z 1005.477,A -85,B 0,C 180,E1 -8891.721,E2 -8891.721} C_VEL
LIN {X 0,Y 553.657,Z 1015.715,A -85,B 0,C 180,E1 -8893.96,E2 -8893.96} C_VEL
LIN {X 0,Y 552.902,Z 1024.892,A -85,B 0,C 180,E1 -8896.296,E2 -8896.296} C_VEL
LIN {X 0,Y 552.381,Z 1032.631,A -85,B 0,C 180,E1 -8898.726,E2 -8898.726} C_VEL
LIN {X 0,Y 552.112,Z 1038.349,A -85,B 0,C 180,E1 -8900.935,E2 -8900.935} C_VEL
LIN {X 0,Y 551.971,Z 1043.475,A -85,B 0,C 180,E1 -8903.551,E2 -8903.551} C_VEL
LIN {X 0,Y 551.929,Z 1046.39,A -85,B 0,C 180,E1 -8905.74,E2 -8905.74} C_VEL
LIN {X 0,Y 551.913,Z 1048.227,A -85,B 0,C 180,E1 -8908.027,E2 -8908.027} C_VEL
LIN {X 0,Y 551.899,Z 1048.659,A -85,B 0,C 180,E1 -8910.623,E2 -8910.623} C_VEL
LIN {X 0,Y 551.907,Z 1047.817,A -85,B 0,C 180,E1 -8912.7,E2 -8912.7} C_VEL
LIN {X 0,Y 551.935,Z 1045.595,A -85,B 0,C 180,E1 -8915.093,E2 -8915.093} C_VEL
LIN {X 0,Y 552.003,Z 1041.594,A -85,B 0,C 180,E1 -8917.599,E2 -8917.599} C_VEL
LIN {X 0,Y 552.188,Z 1036.812,A -85,B 0,C 180,E1 -8919.8,E2 -8919.8} C_VEL
LIN {X 0,Y 552.59,Z 1029.413,A -85,B 0,C 180,E1 -8922.435,E2 -8922.435} C_VEL
LIN {X 0,Y 553.147,Z 1021.637,A -85,B 0,C 180,E1 -8924.659,E2 -8924.659} C_VEL
LIN {X 0,Y 554.083,Z 1011.477,A -85,B 0,C 180,E1 -8927.107,E2 -8927.107} C_VEL
LIN {X 0,Y 555.266,Z 1000.361,A -85,B 0,C 180,E1 -8929.35,E2 -8929.35} C_VEL
LIN {X 0,Y 556.848,Z 987.579,A -85,B 0,C 180,E1 -8931.599,E2 -8931.599} C_VEL
LIN {X 0,Y 558.759,Z 973.271,A -85,B 0,C 180,E1 -8933.743,E2 -8933.743} C_VEL
LIN {X 0,Y 560.976,Z 957.867,A -85,B 0,C 180,E1 -8935.78,E2 -8935.78} C_VEL
LIN {X 0,Y 563.463,Z 940.906,A -85,B 0,C 180,E1 -8937.706,E2 -8937.706} C_VEL
LIN {X 0,Y 566.054,Z 923.597,A -85,B 0,C 180,E1 -8939.442,E2 -8939.442} C_VEL
LIN {X 0,Y 568.921,Z 903.946,A -85,B 0,C 180,E1 -8941.139,E2 -8941.139} C_VEL
LIN {X 0,Y 571.537,Z 885.709,A -85,B 0,C 180,E1 -8942.515,E2 -8942.515} C_VEL
LIN {X 0,Y 574.388,Z 864.383,A -85,B 0,C 180,E1 -8943.9,E2 -8943.9} C_VEL
LIN {X 0,Y 576.71,Z 845.378,A -85,B 0,C 180,E1 -8944.961,E2 -8944.961} C_VEL
LIN {X 0,Y 579.214,Z 823.557,A -85,B 0,C 180,E1 -8946.001,E2 -8946.001} C_VEL
LIN {X 0,Y 581.363,Z 800.758,A -85,B 0,C 180,E1 -8946.888,E2 -8946.888} C_VEL
LIN {X 0,Y 583.363,Z 777.002,A -85,B 0,C 180,E1 -8947.634,E2 -8947.634} C_VEL
LIN {X 0,Y 584.811,Z 753.599,A -85,B 0,C 180,E1 -8948.18,E2 -8948.18} C_VEL
LIN {X 0,Y 585.796,Z 730.838,A -85,B 0,C 180,E1 -8948.572,E2 -8948.572} C_VEL
LIN {X 0,Y 592.182,Z 477.271,A -85,B 0,C 180,E1 -8952.03,E2 -8952.03} C_VEL
LIN {X 0,Y 593.713,Z 414.103,A -85,B 0,C 180,E1 -8952.913,E2 -8952.913} C_VEL
LIN {X 0,Y 579.721,Z 391.22,A -85,B 0,C 180,E1 -8954.61,E2 -8954.61} C_VEL
LIN {X 0,Y 567.964,Z 373.433,A -85,B 0,C 180,E1 -8956.117,E2 -8956.117} C_VEL
LIN {X 0,Y 563.68,Z 367.483,A -85,B 0,C 180,E1 -8956.682,E2 -8956.682} C_VEL
LIN {X 0,Y 560.194,Z 362.701,A -85,B 0,C 180,E1 -8957.152,E2 -8957.152} C_VEL
LIN {X 0,Y 557.505,Z 358.815,A -85,B 0,C 180,E1 -8957.526,E2 -8957.526} C_VEL
LIN {X 0,Y 556.604,Z 357.629,A -85,B 0,C 180,E1 -8957.65,E2 -8957.65} C_VEL
LIN {X 0,Y 554.263,Z 354.846,A -85,B 0,C 180,E1 -8957.971,E2 -8957.971} C_VEL
LIN {X 0,Y 553.454,Z 352.238,A -85,B 0,C 180,E1 -8958.151,E2 -8958.151} C_VEL
LIN {X 0,Y 553.465,Z 352.29,A -85,B 0,C 180,E1 -8961.179,E2 -8961.179} C_VEL
LIN {X 0,Y 553.444,Z 352.291,A -85,B 0,C 180,E1 -8964.553,E2 -8964.553} C_VEL
LIN {X 0,Y 553.504,Z 352.28,A -85,B 0,C 180,E1 -8967.798,E2 -8967.798} C_VEL
LIN {X 0,Y 553.444,Z 352.292,A -85,B 0,C 180,E1 -8970.977,E2 -8970.977} C_VEL
LIN {X 0,Y 553.469,Z 352.288,A -85,B 0,C 180,E1 -8974.305,E2 -8974.305} C_VEL
LIN {X 0,Y 553.467,Z 352.28,A -85,B 0,C 180,E1 -8977.48,E2 -8977.48} C_VEL
LIN {X 0,Y 553.444,Z 352.275,A -85,B 0,C 180,E1 -8980.803,E2 -8980.803} C_VEL
LIN {X 0,Y 553.503,Z 352.266,A -85,B 0,C 180,E1 -8984.063,E2 -8984.063} C_VEL
LIN {X 0,Y 553.443,Z 352.29,A -85,B 0,C 180,E1 -8987.267,E2 -8987.267} C_VEL
LIN {X 0,Y 553.464,Z 352.287,A -85,B 0,C 180,E1 -8990.642,E2 -8990.642} C_VEL
LIN {X 0,Y 553.455,Z 352.27,A -85,B 0,C 180,E1 -8993.673,E2 -8993.673} C_VEL
LIN {X 0,Y 553.445,Z 352.285,A -85,B 0,C 180,E1 -8996.997,E2 -8996.997} C_VEL
LIN {X 0,Y 553.506,Z 352.281,A -85,B 0,C 180,E1 -9000.207,E2 -9000.207} C_VEL
LIN {X 0,Y 553.437,Z 352.268,A -85,B 0,C 180,E1 -9003.418,E2 -9003.418} C_VEL
LIN {X 0,Y 553.491,Z 352.273,A -85,B 0,C 180,E1 -9006.639,E2 -9006.639} C_VEL
LIN {X 0,Y 553.446,Z 352.289,A -85,B 0,C 180,E1 -9009.778,E2 -9009.778} C_VEL
LIN {X 0,Y 553.445,Z 352.282,A -85,B 0,C 180,E1 -9013.265,E2 -9013.265} C_VEL
LIN {X 0,Y 553.491,Z 352.267,A -85,B 0,C 180,E1 -9016.411,E2 -9016.411} C_VEL
LIN {X 0,Y 553.439,Z 352.285,A -85,B 0,C 180,E1 -9019.636,E2 -9019.636} C_VEL
LIN {X 0,Y 553.496,Z 352.282,A -85,B 0,C 180,E1 -9022.881,E2 -9022.881} C_VEL
LIN {X 0,Y 553.451,Z 352.288,A -85,B 0,C 180,E1 -9026.116,E2 -9026.116} C_VEL
LIN {X 0,Y 553.448,Z 352.291,A -85,B 0,C 180,E1 -9029.552,E2 -9029.552} C_VEL
LIN {X 0,Y 553.492,Z 352.287,A -85,B 0,C 180,E1 -9032.694,E2 -9032.694} C_VEL
LIN {X 0,Y 553.44,Z 352.294,A -85,B 0,C 180,E1 -9035.963,E2 -9035.963} C_VEL
LIN {X 0,Y 553.486,Z 352.264,A -85,B 0,C 180,E1 -9039.219,E2 -9039.219} C_VEL
LIN {X 0,Y 553.451,Z 352.322,A -85,B 0,C 180,E1 -9039.679,E2 -9039.679} C_VEL
LIN {X 0,Y 554.631,Z 355.561,A -85,B 0,C 180,E1 -9040.196,E2 -9040.196} C_VEL
LIN {X 0,Y 558.837,Z 364.98,A -85,B 0,C 180,E1 -9041.745,E2 -9041.745} C_VEL
LIN {X 0,Y 562.177,Z 372.698,A -85,B 0,C 180,E1 -9042.919,E2 -9042.919} C_VEL
LIN {X 0,Y 574.778,Z 392.017,A -85,B 0,C 180,E1 -9044.583,E2 -9044.583} C_VEL
LIN {X 0,Y 588.135,Z 414.181,A -85,B 0,C 180,E1 -9046.248,E2 -9046.248} C_VEL
LIN {X 0,Y 593.82,Z 424.386,A -85,B 0,C 180,E1 -9046.933,E2 -9046.933} C_VEL
LIN {X 0,Y 587.198,Z 685.756,A -85,B 0,C 180,E1 -9050.506,E2 -9050.506} C_VEL
LIN {X 0,Y 585.11,Z 765.891,A -85,B 0,C 180,E1 -9051.613,E2 -9051.613} C_VEL
LIN {X 0,Y 583.597,Z 791.529,A -85,B 0,C 180,E1 -9052.128,E2 -9052.128} C_VEL
LIN {X 0,Y 581.925,Z 813.462,A -85,B 0,C 180,E1 -9052.722,E2 -9052.722} C_VEL
LIN {X 0,Y 579.757,Z 837.297,A -85,B 0,C 180,E1 -9053.548,E2 -9053.548} C_VEL
LIN {X 0,Y 577.556,Z 858.023,A -85,B 0,C 180,E1 -9054.43,E2 -9054.43} C_VEL
LIN {X 0,Y 574.976,Z 880.16,A -85,B 0,C 180,E1 -9055.542,E2 -9055.542} C_VEL
LIN {X 0,Y 572.174,Z 901.61,A -85,B 0,C 180,E1 -9056.832,E2 -9056.832} C_VEL
LIN {X 0,Y 569.384,Z 922.313,A -85,B 0,C 180,E1 -9058.268,E2 -9058.268} C_VEL
LIN {X 0,Y 566.607,Z 941.752,A -85,B 0,C 180,E1 -9059.849,E2 -9059.849} C_VEL
LIN {X 0,Y 564.034,Z 959.851,A -85,B 0,C 180,E1 -9061.519,E2 -9061.519} C_VEL
LIN {X 0,Y 561.434,Z 977.933,A -85,B 0,C 180,E1 -9063.447,E2 -9063.447} C_VEL
LIN {X 0,Y 559.367,Z 993.031,A -85,B 0,C 180,E1 -9065.274,E2 -9065.274} C_VEL
LIN {X 0,Y 557.247,Z 1009.268,A -85,B 0,C 180,E1 -9067.532,E2 -9067.532} C_VEL
LIN {X 0,Y 555.718,Z 1022.047,A -85,B 0,C 180,E1 -9069.57,E2 -9069.57} C_VEL
LIN {X 0,Y 554.314,Z 1035.356,A -85,B 0,C 180,E1 -9072.034,E2 -9072.034} C_VEL
LIN {X 0,Y 553.459,Z 1044.765,A -85,B 0,C 180,E1 -9074.061,E2 -9074.061} C_VEL
LIN {X 0,Y 552.75,Z 1054.482,A -85,B 0,C 180,E1 -9076.505,E2 -9076.505} C_VEL
LIN {X 0,Y 552.313,Z 1061.983,A -85,B 0,C 180,E1 -9078.831,E2 -9078.831} C_VEL
LIN {X 0,Y 552.061,Z 1068.076,A -85,B 0,C 180,E1 -9081.144,E2 -9081.144} C_VEL
LIN {X 0,Y 551.95,Z 1072.983,A -85,B 0,C 180,E1 -9083.655,E2 -9083.655} C_VEL
LIN {X 0,Y 551.916,Z 1075.819,A -85,B 0,C 180,E1 -9085.74,E2 -9085.74} C_VEL
LIN {X 0,Y 551.907,Z 1077.7,A -85,B 0,C 180,E1 -9088.027,E2 -9088.027} C_VEL
LIN {X 0,Y 551.899,Z 1078.132,A -85,B 0,C 180,E1 -9090.519,E2 -9090.519} C_VEL
LIN {X 0,Y 551.91,Z 1077.216,A -85,B 0,C 180,E1 -9092.7,E2 -9092.7} C_VEL
LIN {X 0,Y 551.933,Z 1074.892,A -85,B 0,C 180,E1 -9095.093,E2 -9095.093} C_VEL
LIN {X 0,Y 551.985,Z 1070.924,A -85,B 0,C 180,E1 -9097.494,E2 -9097.494} C_VEL
LIN {X 0,Y 552.143,Z 1066.009,A -85,B 0,C 180,E1 -9099.696,E2 -9099.696} C_VEL
LIN {X 0,Y 552.484,Z 1058.765,A -85,B 0,C 180,E1 -9102.231,E2 -9102.231} C_VEL
LIN {X 0,Y 552.99,Z 1050.856,A -85,B 0,C 180,E1 -9104.449,E2 -9104.449} C_VEL
LIN {X 0,Y 553.8,Z 1041.047,A -85,B 0,C 180,E1 -9106.791,E2 -9106.791} C_VEL
LIN {X 0,Y 554.932,Z 1029.257,A -85,B 0,C 180,E1 -9109.143,E2 -9109.143} C_VEL
LIN {X 0,Y 556.316,Z 1016.907,A -85,B 0,C 180,E1 -9111.288,E2 -9111.288} C_VEL
LIN {X 0,Y 558.196,Z 1001.817,A -85,B 0,C 180,E1 -9113.544,E2 -9113.544} C_VEL
LIN {X 0,Y 560.083,Z 987.687,A -85,B 0,C 180,E1 -9115.399,E2 -9115.399} C_VEL
LIN {X 0,Y 562.685,Z 969.174,A -85,B 0,C 180,E1 -9117.517,E2 -9117.517} C_VEL
LIN {X 0,Y 565.047,Z 952.568,A -85,B 0,C 180,E1 -9119.177,E2 -9119.177} C_VEL
LIN {X 0,Y 568.032,Z 931.716,A -85,B 0,C 180,E1 -9120.99,E2 -9120.99} C_VEL
LIN {X 0,Y 570.483,Z 914.166,A -85,B 0,C 180,E1 -9122.315,E2 -9122.315} C_VEL
LIN {X 0,Y 573.329,Z 893.112,A -85,B 0,C 180,E1 -9123.706,E2 -9123.706} C_VEL
LIN {X 0,Y 575.911,Z 871.844,A -85,B 0,C 180,E1 -9124.895,E2 -9124.895} C_VEL
LIN {X 0,Y 578.45,Z 850.038,A -85,B 0,C 180,E1 -9125.934,E2 -9125.934} C_VEL
LIN {X 0,Y 580.672,Z 827.403,A -85,B 0,C 180,E1 -9126.815,E2 -9126.815} C_VEL
LIN {X 0,Y 582.529,Z 806.108,A -85,B 0,C 180,E1 -9127.492,E2 -9127.492} C_VEL
LIN {X 0,Y 584.32,Z 780.702,A -85,B 0,C 180,E1 -9128.109,E2 -9128.109} C_VEL
LIN {X 0,Y 585.358,Z 758.863,A -85,B 0,C 180,E1 -9128.492,E2 -9128.492} C_VEL
LIN {X 0,Y 591.364,Z 516.91,A -85,B 0,C 180,E1 -9131.794,E2 -9131.794} C_VEL
LIN {X 0,Y 593.666,Z 423.829,A -85,B 0,C 180,E1 -9133.085,E2 -9133.085} C_VEL
LIN {X 0,Y 580.254,Z 400.889,A -85,B 0,C 180,E1 -9134.716,E2 -9134.716} C_VEL
LIN {X 0,Y 565.909,Z 378.276,A -85,B 0,C 180,E1 -9136.567,E2 -9136.567} C_VEL
LIN {X 0,Y 561.804,Z 371.853,A -85,B 0,C 180,E1 -9137.166,E2 -9137.166} C_VEL
LIN {X 0,Y 556.066,Z 358.788,A -85,B 0,C 180,E1 -9139.252,E2 -9139.252} C_VEL
LIN {X 0,Y 554.587,Z 355.515,A -85,B 0,C 180,E1 -9139.8,E2 -9139.8} C_VEL
LIN {X 0,Y 553.448,Z 352.278,A -85,B 0,C 180,E1 -9140.321,E2 -9140.321} C_VEL
LIN {X 0,Y 553.447,Z 352.229,A -85,B 0,C 180,E1 -9143.684,E2 -9143.684} C_VEL
LIN {X 0,Y 553.492,Z 352.277,A -85,B 0,C 180,E1 -9146.936,E2 -9146.936} C_VEL
LIN {X 0,Y 553.442,Z 352.287,A -85,B 0,C 180,E1 -9150.209,E2 -9150.209} C_VEL
LIN {X 0,Y 553.495,Z 352.276,A -85,B 0,C 180,E1 -9153.408,E2 -9153.408} C_VEL
LIN {X 0,Y 553.45,Z 352.278,A -85,B 0,C 180,E1 -9156.603,E2 -9156.603} C_VEL
LIN {X 0,Y 553.45,Z 352.274,A -85,B 0,C 180,E1 -9160.034,E2 -9160.034} C_VEL
LIN {X 0,Y 553.493,Z 352.273,A -85,B 0,C 180,E1 -9163.226,E2 -9163.226} C_VEL
LIN {X 0,Y 553.442,Z 352.288,A -85,B 0,C 180,E1 -9166.416,E2 -9166.416} C_VEL
LIN {X 0,Y 553.494,Z 352.279,A -85,B 0,C 180,E1 -9169.698,E2 -9169.698} C_VEL
LIN {X 0,Y 553.445,Z 352.266,A -85,B 0,C 180,E1 -9172.839,E2 -9172.839} C_VEL
LIN {X 0,Y 553.454,Z 352.278,A -85,B 0,C 180,E1 -9176.271,E2 -9176.271} C_VEL
LIN {X 0,Y 553.494,Z 352.283,A -85,B 0,C 180,E1 -9179.482,E2 -9179.482} C_VEL
LIN {X 0,Y 553.441,Z 352.275,A -85,B 0,C 180,E1 -9182.692,E2 -9182.692} C_VEL
LIN {X 0,Y 553.502,Z 352.269,A -85,B 0,C 180,E1 -9185.91,E2 -9185.91} C_VEL
LIN {X 0,Y 553.446,Z 352.289,A -85,B 0,C 180,E1 -9189.043,E2 -9189.043} C_VEL
LIN {X 0,Y 553.465,Z 352.277,A -85,B 0,C 180,E1 -9192.415,E2 -9192.415} C_VEL
LIN {X 0,Y 553.467,Z 352.271,A -85,B 0,C 180,E1 -9195.508,E2 -9195.508} C_VEL
LIN {X 0,Y 553.448,Z 352.283,A -85,B 0,C 180,E1 -9198.868,E2 -9198.868} C_VEL
LIN {X 0,Y 553.513,Z 352.284,A -85,B 0,C 180,E1 -9202.073,E2 -9202.073} C_VEL
LIN {X 0,Y 553.45,Z 352.287,A -85,B 0,C 180,E1 -9205.352,E2 -9205.352} C_VEL
LIN {X 0,Y 553.467,Z 352.28,A -85,B 0,C 180,E1 -9208.722,E2 -9208.722} C_VEL
LIN {X 0,Y 553.48,Z 352.271,A -85,B 0,C 180,E1 -9211.889,E2 -9211.889} C_VEL
LIN {X 0,Y 553.449,Z 352.28,A -85,B 0,C 180,E1 -9215.193,E2 -9215.193} C_VEL
LIN {X 0,Y 553.509,Z 352.274,A -85,B 0,C 180,E1 -9218.42,E2 -9218.42} C_VEL
LIN {X 0,Y 553.455,Z 352.293,A -85,B 0,C 180,E1 -9221.67,E2 -9221.67} C_VEL
LIN {X 0,Y 553.506,Z 352.498,A -85,B 0,C 180,E1 -9222,E2 -9222} C_VEL
LIN {X 0,Y 554.715,Z 355.633,A -85,B 0,C 180,E1 -9222.199,E2 -9222.199} C_VEL
LIN {X 0,Y 557.373,Z 358.543,A -85,B 0,C 180,E1 -9222.557,E2 -9222.557} C_VEL
LIN {X 0,Y 560.052,Z 362.56,A -85,B 0,C 180,E1 -9222.931,E2 -9222.931} C_VEL
LIN {X 0,Y 561.722,Z 364.777,A -85,B 0,C 180,E1 -9223.156,E2 -9223.156} C_VEL
LIN {X 0,Y 567.756,Z 373.138,A -85,B 0,C 180,E1 -9223.956,E2 -9223.956} C_VEL
LIN {X 0,Y 579.755,Z 391.291,A -85,B 0,C 180,E1 -9225.492,E2 -9225.492} C_VEL
LIN {X 0,Y 593.78,Z 414.26,A -85,B 0,C 180,E1 -9227.191,E2 -9227.191} C_VEL
LIN {X 0,Y 587.558,Z 658.694,A -85,B 0,C 180,E1 -9230.539,E2 -9230.539} C_VEL
LIN {X 0,Y 586.911,Z 685.209,A -85,B 0,C 180,E1 -9230.898,E2 -9230.898} C_VEL
LIN {X 0,Y 585.947,Z 692.902,A -85,B 0,C 180,E1 -9230.94,E2 -9230.94} C_VEL
LIN {X 0,Y 580.621,Z 713.438,A -85,B 0,C 180,E1 -9230.832,E2 -9230.832} C_VEL
LIN {X 0,Y 579.851,Z 720.042,A -85,B 0,C 180,E1 -9230.873,E2 -9230.873} C_VEL
LIN {X 0,Y 578.718,Z 750.314,A -85,B 0,C 180,E1 -9231.353,E2 -9231.353} C_VEL
LIN {X 0,Y 577.444,Z 770.755,A -85,B 0,C 180,E1 -9231.809,E2 -9231.809} C_VEL
LIN {X 0,Y 575.602,Z 794.348,A -85,B 0,C 180,E1 -9232.493,E2 -9232.493} C_VEL
LIN {X 0,Y 573.465,Z 816.188,A -85,B 0,C 180,E1 -9233.305,E2 -9233.305} C_VEL
